LIN {X 85.009,Y 2.500,Z 47.262,A 180.000,B 0.000,C 180.000} C_DIS
LIN {X 84.772,Y 2.500,Z 47.254,A 180.000,B 0.000,C 180.000} C_DIS
LIN {X 84.615,Y 2.500,Z 47.248,A 180.000,B 0.000,C 180.000} C_DIS
LIN {X 84.536,Y 2.500,Z 47.246,A 180.000,B 0.000,C 180.000} C_DIS
LIN {X 84.379,Y 2.500,Z 47.240,A 180.000,B 0.000,C 180.000} C_DIS
LIN {X 84.142,Y 2.500,Z 47.232,A 180.000,B 0.000,C 180.000} C_DIS
LIN {X 83.985,Y 2.500,Z 47.226,A 180.000,B 0.000,C 180.000} C_DIS
LIN {X 83.906,Y 2.500,Z 47.224,A 180.000,B 0.000,C 180.000} C_DIS
LIN {X 83.749,Y 2.500,Z 47.218,A 180.000,B 0.000,C 180.000} C_DIS
LIN {X 83.512,Y 2.500,Z 47.210,A 180.000,B 0.000,C 180.000} C_DIS
LIN {X 83.355,Y 2.500,Z 47.204,A 180.000,B 0.000,C 180.000} C_DIS
LIN {X 83.276,Y 2.500,Z 47.202,A 180.000,B 0.000,C 180.000} C_DIS
LIN {X 83.119,Y 2.500,Z 47.196,A 180.000,B 0.000,C 180.000} C_DIS
LIN {X 82.961,Y 2.500,Z 47.191,A 180.000,B 0.000,C 180.000} C_DIS
LIN {X 82.804,Y 2.500,Z 47.185,A 180.000,B 0.000,C 180.000} C_DIS
LIN {X 82.646,Y 2.500,Z 47.180,A 180.000,B 0.000,C 180.000} C_DIS
LIN {X 82.489,Y 2.500,Z 47.174,A 180.000,B 0.000,C 180.000} C_DIS
LIN {X 82.331,Y 2.500,Z 47.169,A 180.000,B 0.000,C 180.000} C_DIS
LIN {X 82.174,Y 2.500,Z 47.164,A 180.000,B 0.000,C 180.000} C_DIS
LIN {X 82.095,Y 2.500,Z 47.161,A 180.000,B 0.000,C 180.000} C_DIS
LIN {X 82.016,Y 2.500,Z 47.159,A 180.000,B 0.000,C 180.000} C_DIS
LIN {X 81.937,Y 2.500,Z 47.156,A 180.000,B 0.000,C 180.000} C_DIS
LIN {X 81.859,Y 2.500,Z 47.154,A 180.000,B 0.000,C 180.000} C_DIS
LIN {X 81.780,Y 2.500,Z 47.151,A 180.000,B 0.000,C 180.000} C_DIS
LIN {X 81.701,Y 2.500,Z 47.148,A 180.000,B 0.000,C 180.000} C_DIS
LIN {X 81.544,Y 2.500,Z 47.143,A 180.000,B 0.000,C 180.000} C_DIS
LIN {X 81.386,Y 2.500,Z 47.139,A 180.000,B 0.000,C 180.000} C_DIS
LIN {X 81.229,Y 2.500,Z 47.134,A 180.000,B 0.000,C 180.000} C_DIS
LIN {X 81.071,Y 2.500,Z 47.129,A 180.000,B 0.000,C 180.000} C_DIS
LIN {X 80.914,Y 2.500,Z 47.124,A 180.000,B 0.000,C 180.000} C_DIS
LIN {X 80.756,Y 2.500,Z 47.120,A 180.000,B 0.000,C 180.000} C_DIS
LIN {X 80.599,Y 2.500,Z 47.115,A 180.000,B 0.000,C 180.000} C_DIS
LIN {X 80.441,Y 2.500,Z 47.110,A 180.000,B 0.000,C 180.000} C_DIS
LIN {X 80.284,Y 2.500,Z 47.106,A 180.000,B 0.000,C 180.000} C_DIS
LIN {X 80.126,Y 2.500,Z 47.102,A 180.000,B 0.000,C 180.000} C_DIS
LIN {X 79.969,Y 2.500,Z 47.097,A 180.000,B 0.000,C 180.000} C_DIS
LIN {X 79.811,Y 2.500,Z 47.093,A 180.000,B 0.000,C 180.000} C_DIS
LIN {X 79.654,Y 2.500,Z 47.089,A 180.000,B 0.000,C 180.000} C_DIS
LIN {X 79.496,Y 2.500,Z 47.085,A 180.000,B 0.000,C 180.000} C_DIS
LIN {X 79.339,Y 2.500,Z 47.081,A 180.000,B 0.000,C 180.000} C_DIS
LIN {X 79.181,Y 2.500,Z 47.077,A 180.000,B 0.000,C 180.000} C_DIS
LIN {X 79.024,Y 2.500,Z 47.073,A 180.000,B 0.000,C 180.000} C_DIS
LIN {X 78.866,Y 2.500,Z 47.070,A 180.000,B 0.000,C 180.000} C_DIS
LIN {X 78.709,Y 2.500,Z 47.066,A 180.000,B 0.000,C 180.000} C_DIS
LIN {X 78.551,Y 2.500,Z 47.062,A 180.000,B 0.000,C 180.000} C_DIS
LIN {X 78.394,Y 2.500,Z 47.059,A 180.000,B 0.000,C 180.000} C_DIS
LIN {X 78.236,Y 2.500,Z 47.056,A 180.000,B 0.000,C 180.000} C_DIS
LIN {X 78.079,Y 2.500,Z 47.052,A 180.000,B 0.000,C 180.000} C_DIS
LIN {X 77.921,Y 2.500,Z 47.049,A 180.000,B 0.000,C 180.000} C_DIS
LIN {X 77.764,Y 2.500,Z 47.046,A 180.000,B 0.000,C 180.000} C_DIS
LIN {X 77.606,Y 2.500,Z 47.043,A 180.000,B 0.000,C 180.000} C_DIS
LIN {X 77.449,Y 2.500,Z 47.040,A 180.000,B 0.000,C 180.000} C_DIS
LIN {X 77.291,Y 2.500,Z 47.037,A 180.000,B 0.000,C 180.000} C_DIS
LIN {X 77.134,Y 2.500,Z 47.034,A 180.000,B 0.000,C 180.000} C_DIS
LIN {X 76.976,Y 2.500,Z 47.032,A 180.000,B 0.000,C 180.000} C_DIS
LIN {X 76.819,Y 2.500,Z 47.029,A 180.000,B 0.000,C 180.000} C_DIS
LIN {X 76.661,Y 2.500,Z 47.027,A 180.000,B 0.000,C 180.000} C_DIS
LIN {X 76.346,Y 2.500,Z 47.022,A 180.000,B 0.000,C 180.000} C_DIS
LIN {X 76.031,Y 2.500,Z 47.018,A 180.000,B 0.000,C 180.000} C_DIS
LIN {X 75.716,Y 2.500,Z 47.014,A 180.000,B 0.000,C 180.000} C_DIS
LIN {X 75.401,Y 2.500,Z 47.011,A 180.000,B 0.000,C 180.000} C_DIS
LIN {X 75.086,Y 2.500,Z 47.008,A 180.000,B 0.000,C 180.000} C_DIS
LIN {X 74.771,Y 2.500,Z 47.005,A 180.000,B 0.000,C 180.000} C_DIS
LIN {X 74.456,Y 2.500,Z 47.003,A 180.000,B 0.000,C 180.000} C_DIS
LIN {X 74.141,Y 2.500,Z 47.002,A 180.000,B 0.000,C 180.000} C_DIS
LIN {X 73.826,Y 2.500,Z 47.001,A 180.000,B 0.000,C 180.000} C_DIS
LIN {X 73.511,Y 2.500,Z 47.000,A 180.000,B 0.000,C 180.000} C_DIS
LIN {X 73.280,Y 2.500,Z 47.000,A 180.000,B 0.000,C 180.000} C_DIS
; Cutting Move Starts
LIN {X 5.009,Y 2.500,Z 47.000,A 180.000,B 0.000,C 180.000} C_DIS
LIN {X 4.830,Y 2.506,Z 47.000,A 180.000,B 0.000,C 180.000} C_DIS
LIN {X 4.827,Y 2.506,Z 47.000,A 180.000,B 0.000,C 180.000} C_DIS
LIN {X 4.651,Y 2.524,Z 47.000,A 180.000,B 0.000,C 180.000} C_DIS
LIN {X 4.472,Y 2.556,Z 47.000,A 180.000,B 0.000,C 180.000} C_DIS
LIN {X 4.294,Y 2.602,Z 47.000,A 180.000,B 0.000,C 180.000} C_DIS
LIN {X 4.115,Y 2.662,Z 47.000,A 180.000,B 0.000,C 180.000} C_DIS
LIN {X 4.057,Y 2.685,Z 47.000,A 180.000,B 0.000,C 180.000} C_DIS
LIN {X 3.936,Y 2.738,Z 47.000,A 180.000,B 0.000,C 180.000} C_DIS
LIN {X 3.757,Y 2.831,Z 47.000,A 180.000,B 0.000,C 180.000} C_DIS
LIN {X 3.702,Y 2.864,Z 47.000,A 180.000,B 0.000,C 180.000} C_DIS
LIN {X 3.579,Y 2.943,Z 47.000,A 180.000,B 0.000,C 180.000} C_DIS
LIN {X 3.445,Y 3.042,Z 47.000,A 180.000,B 0.000,C 180.000} C_DIS
LIN {X 3.400,Y 3.079,Z 47.000,A 180.000,B 0.000,C 180.000} C_DIS
LIN {X 3.243,Y 3.221,Z 47.000,A 180.000,B 0.000,C 180.000} C_DIS
LIN {X 3.221,Y 3.243,Z 47.000,A 180.000,B 0.000,C 180.000} C_DIS
LIN {X 3.079,Y 3.400,Z 47.000,A 180.000,B 0.000,C 180.000} C_DIS
LIN {X 3.042,Y 3.445,Z 47.000,A 180.000,B 0.000,C 180.000} C_DIS
LIN {X 2.943,Y 3.579,Z 47.000,A 180.000,B 0.000,C 180.000} C_DIS
LIN {X 2.864,Y 3.702,Z 47.000,A 180.000,B 0.000,C 180.000} C_DIS
LIN {X 2.831,Y 3.757,Z 47.000,A 180.000,B 0.000,C 180.000} C_DIS
LIN {X 2.738,Y 3.936,Z 47.000,A 180.000,B 0.000,C 180.000} C_DIS
LIN {X 2.685,Y 4.057,Z 47.000,A 180.000,B 0.000,C 180.000} C_DIS
LIN {X 2.662,Y 4.115,Z 47.000,A 180.000,B 0.000,C 180.000} C_DIS
LIN {X 2.602,Y 4.294,Z 47.000,A 180.000,B 0.000,C 180.000} C_DIS
LIN {X 2.556,Y 4.472,Z 47.000,A 180.000,B 0.000,C 180.000} C_DIS
LIN {X 2.524,Y 4.651,Z 47.000,A 180.000,B 0.000,C 180.000} C_DIS
LIN {X 2.506,Y 4.827,Z 47.000,A 180.000,B 0.000,C 180.000} C_DIS
LIN {X 2.506,Y 4.830,Z 47.000,A 180.000,B 0.000,C 180.000} C_DIS
LIN {X 2.500,Y 5.009,Z 47.000,A 180.000,B 0.000,C 180.000} C_DIS
LIN {X 2.500,Y 149.991,Z 47.000,A 180.000,B 0.000,C 180.000} C_DIS
LIN {X 2.506,Y 150.170,Z 47.000,A 180.000,B 0.000,C 180.000} C_DIS
LIN {X 2.506,Y 150.173,Z 47.000,A 180.000,B 0.000,C 180.000} C_DIS
LIN {X 2.524,Y 150.349,Z 47.000,A 180.000,B 0.000,C 180.000} C_DIS
LIN {X 2.556,Y 150.528,Z 47.000,A 180.000,B 0.000,C 180.000} C_DIS
LIN {X 2.602,Y 150.706,Z 47.000,A 180.000,B 0.000,C 180.000} C_DIS
LIN {X 2.662,Y 150.885,Z 47.000,A 180.000,B 0.000,C 180.000} C_DIS
LIN {X 2.685,Y 150.943,Z 47.000,A 180.000,B 0.000,C 180.000} C_DIS
LIN {X 2.738,Y 151.064,Z 47.000,A 180.000,B 0.000,C 180.000} C_DIS
LIN {X 2.831,Y 151.243,Z 47.000,A 180.000,B 0.000,C 180.000} C_DIS
LIN {X 2.864,Y 151.298,Z 47.000,A 180.000,B 0.000,C 180.000} C_DIS
LIN {X 2.943,Y 151.421,Z 47.000,A 180.000,B 0.000,C 180.000} C_DIS
LIN {X 3.042,Y 151.555,Z 47.000,A 180.000,B 0.000,C 180.000} C_DIS
LIN {X 3.079,Y 151.600,Z 47.000,A 180.000,B 0.000,C 180.000} C_DIS
LIN {X 3.221,Y 151.757,Z 47.000,A 180.000,B 0.000,C 180.000} C_DIS
LIN {X 3.243,Y 151.779,Z 47.000,A 180.000,B 0.000,C 180.000} C_DIS
LIN {X 3.400,Y 151.921,Z 47.000,A 180.000,B 0.000,C 180.000} C_DIS
LIN {X 3.445,Y 151.958,Z 47.000,A 180.000,B 0.000,C 180.000} C_DIS
LIN {X 3.579,Y 152.057,Z 47.000,A 180.000,B 0.000,C 180.000} C_DIS
LIN {X 3.702,Y 152.136,Z 47.000,A 180.000,B 0.000,C 180.000} C_DIS
LIN {X 3.757,Y 152.169,Z 47.000,A 180.000,B 0.000,C 180.000} C_DIS
LIN {X 3.936,Y 152.262,Z 47.000,A 180.000,B 0.000,C 180.000} C_DIS
LIN {X 4.057,Y 152.315,Z 47.000,A 180.000,B 0.000,C 180.000} C_DIS
LIN {X 4.115,Y 152.338,Z 47.000,A 180.000,B 0.000,C 180.000} C_DIS
LIN {X 4.294,Y 152.398,Z 47.000,A 180.000,B 0.000,C 180.000} C_DIS
LIN {X 4.472,Y 152.444,Z 47.000,A 180.000,B 0.000,C 180.000} C_DIS
LIN {X 4.651,Y 152.476,Z 47.000,A 180.000,B 0.000,C 180.000} C_DIS
LIN {X 4.827,Y 152.494,Z 47.000,A 180.000,B 0.000,C 180.000} C_DIS
LIN {X 4.830,Y 152.494,Z 47.000,A 180.000,B 0.000,C 180.000} C_DIS
LIN {X 5.009,Y 152.500,Z 47.000,A 180.000,B 0.000,C 180.000} C_DIS
LIN {X 149.991,Y 152.500,Z 47.000,A 180.000,B 0.000,C 180.000} C_DIS
LIN {X 150.170,Y 152.494,Z 47.000,A 180.000,B 0.000,C 180.000} C_DIS
LIN {X 150.173,Y 152.494,Z 47.000,A 180.000,B 0.000,C 180.000} C_DIS
LIN {X 150.349,Y 152.476,Z 47.000,A 180.000,B 0.000,C 180.000} C_DIS
LIN {X 150.528,Y 152.444,Z 47.000,A 180.000,B 0.000,C 180.000} C_DIS
LIN {X 150.706,Y 152.398,Z 47.000,A 180.000,B 0.000,C 180.000} C_DIS
LIN {X 150.885,Y 152.338,Z 47.000,A 180.000,B 0.000,C 180.000} C_DIS
LIN {X 150.943,Y 152.315,Z 47.000,A 180.000,B 0.000,C 180.000} C_DIS
LIN {X 151.064,Y 152.262,Z 47.000,A 180.000,B 0.000,C 180.000} C_DIS
LIN {X 151.243,Y 152.169,Z 47.000,A 180.000,B 0.000,C 180.000} C_DIS
LIN {X 151.298,Y 152.136,Z 47.000,A 180.000,B 0.000,C 180.000} C_DIS
LIN {X 151.421,Y 152.057,Z 47.000,A 180.000,B 0.000,C 180.000} C_DIS
LIN {X 151.555,Y 151.958,Z 47.000,A 180.000,B 0.000,C 180.000} C_DIS
LIN {X 151.600,Y 151.921,Z 47.000,A 180.000,B 0.000,C 180.000} C_DIS
LIN {X 151.757,Y 151.779,Z 47.000,A 180.000,B 0.000,C 180.000} C_DIS
LIN {X 151.779,Y 151.757,Z 47.000,A 180.000,B 0.000,C 180.000} C_DIS
LIN {X 151.921,Y 151.600,Z 47.000,A 180.000,B 0.000,C 180.000} C_DIS
LIN {X 151.958,Y 151.555,Z 47.000,A 180.000,B 0.000,C 180.000} C_DIS
LIN {X 152.057,Y 151.421,Z 47.000,A 180.000,B 0.000,C 180.000} C_DIS
LIN {X 152.136,Y 151.298,Z 47.000,A 180.000,B 0.000,C 180.000} C_DIS
LIN {X 152.169,Y 151.243,Z 47.000,A 180.000,B 0.000,C 180.000} C_DIS
LIN {X 152.262,Y 151.064,Z 47.000,A 180.000,B 0.000,C 180.000} C_DIS
LIN {X 152.315,Y 150.943,Z 47.000,A 180.000,B 0.000,C 180.000} C_DIS
LIN {X 152.338,Y 150.885,Z 47.000,A 180.000,B 0.000,C 180.000} C_DIS
LIN {X 152.398,Y 150.706,Z 47.000,A 180.000,B 0.000,C 180.000} C_DIS
LIN {X 152.444,Y 150.528,Z 47.000,A 180.000,B 0.000,C 180.000} C_DIS
LIN {X 152.476,Y 150.349,Z 47.000,A 180.000,B 0.000,C 180.000} C_DIS
LIN {X 152.494,Y 150.173,Z 47.000,A 180.000,B 0.000,C 180.000} C_DIS
LIN {X 152.494,Y 150.170,Z 47.000,A 180.000,B 0.000,C 180.000} C_DIS
LIN {X 152.500,Y 149.991,Z 47.000,A 180.000,B 0.000,C 180.000} C_DIS
LIN {X 152.500,Y 5.009,Z 47.000,A 180.000,B 0.000,C 180.000} C_DIS
LIN {X 152.494,Y 4.830,Z 47.000,A 180.000,B 0.000,C 180.000} C_DIS
LIN {X 152.494,Y 4.827,Z 47.000,A 180.000,B 0.000,C 180.000} C_DIS
LIN {X 152.476,Y 4.651,Z 47.000,A 180.000,B 0.000,C 180.000} C_DIS
LIN {X 152.444,Y 4.472,Z 47.000,A 180.000,B 0.000,C 180.000} C_DIS
LIN {X 152.398,Y 4.294,Z 47.000,A 180.000,B 0.000,C 180.000} C_DIS
LIN {X 152.338,Y 4.115,Z 47.000,A 180.000,B 0.000,C 180.000} C_DIS
LIN {X 152.315,Y 4.057,Z 47.000,A 180.000,B 0.000,C 180.000} C_DIS
LIN {X 152.262,Y 3.936,Z 47.000,A 180.000,B 0.000,C 180.000} C_DIS
LIN {X 152.169,Y 3.757,Z 47.000,A 180.000,B 0.000,C 180.000} C_DIS
LIN {X 152.136,Y 3.702,Z 47.000,A 180.000,B 0.000,C 180.000} C_DIS
LIN {X 152.057,Y 3.579,Z 47.000,A 180.000,B 0.000,C 180.000} C_DIS
LIN {X 151.958,Y 3.445,Z 47.000,A 180.000,B 0.000,C 180.000} C_DIS
LIN {X 151.921,Y 3.400,Z 47.000,A 180.000,B 0.000,C 180.000} C_DIS
LIN {X 151.779,Y 3.243,Z 47.000,A 180.000,B 0.000,C 180.000} C_DIS
LIN {X 151.757,Y 3.221,Z 47.000,A 180.000,B 0.000,C 180.000} C_DIS
LIN {X 151.600,Y 3.079,Z 47.000,A 180.000,B 0.000,C 180.000} C_DIS
LIN {X 151.555,Y 3.042,Z 47.000,A 180.000,B 0.000,C 180.000} C_DIS
LIN {X 151.421,Y 2.943,Z 47.000,A 180.000,B 0.000,C 180.000} C_DIS
LIN {X 151.298,Y 2.864,Z 47.000,A 180.000,B 0.000,C 180.000} C_DIS
LIN {X 151.243,Y 2.831,Z 47.000,A 180.000,B 0.000,C 180.000} C_DIS
LIN {X 151.064,Y 2.738,Z 47.000,A 180.000,B 0.000,C 180.000} C_DIS
LIN {X 150.943,Y 2.685,Z 47.000,A 180.000,B 0.000,C 180.000} C_DIS
LIN {X 150.885,Y 2.662,Z 47.000,A 180.000,B 0.000,C 180.000} C_DIS
LIN {X 150.706,Y 2.602,Z 47.000,A 180.000,B 0.000,C 180.000} C_DIS
LIN {X 150.528,Y 2.556,Z 47.000,A 180.000,B 0.000,C 180.000} C_DIS
LIN {X 150.349,Y 2.524,Z 47.000,A 180.000,B 0.000,C 180.000} C_DIS
LIN {X 150.173,Y 2.506,Z 47.000,A 180.000,B 0.000,C 180.000} C_DIS
LIN {X 150.170,Y 2.506,Z 47.000,A 180.000,B 0.000,C 180.000} C_DIS
LIN {X 149.991,Y 2.500,Z 47.000,A 180.000,B 0.000,C 180.000} C_DIS
LIN {X 110.366,Y 2.500,Z 47.000,A 180.000,B 0.000,C 180.000} C_DIS
LIN {X 73.280,Y 2.500,Z 47.000,A 180.000,B 0.000,C 180.000} C_DIS
; Link Move Starts
LIN {X 72.965,Y 2.500,Z 47.000,A 180.000,B 0.000,C 180.000} C_DIS
LIN {X 72.650,Y 2.500,Z 46.999,A 180.000,B 0.000,C 180.000} C_DIS
LIN {X 72.335,Y 2.500,Z 46.998,A 180.000,B 0.000,C 180.000} C_DIS
LIN {X 72.020,Y 2.500,Z 46.996,A 180.000,B 0.000,C 180.000} C_DIS
LIN {X 71.705,Y 2.500,Z 46.994,A 180.000,B 0.000,C 180.000} C_DIS
LIN {X 71.390,Y 2.500,Z 46.991,A 180.000,B 0.000,C 180.000} C_DIS
LIN {X 71.075,Y 2.500,Z 46.988,A 180.000,B 0.000,C 180.000} C_DIS
LIN {X 70.760,Y 2.500,Z 46.985,A 180.000,B 0.000,C 180.000} C_DIS
LIN {X 70.445,Y 2.500,Z 46.981,A 180.000,B 0.000,C 180.000} C_DIS
LIN {X 70.130,Y 2.500,Z 46.977,A 180.000,B 0.000,C 180.000} C_DIS
LIN {X 69.815,Y 2.500,Z 46.972,A 180.000,B 0.000,C 180.000} C_DIS
LIN {X 69.658,Y 2.500,Z 46.969,A 180.000,B 0.000,C 180.000} C_DIS
LIN {X 69.500,Y 2.500,Z 46.967,A 180.000,B 0.000,C 180.000} C_DIS
LIN {X 69.343,Y 2.500,Z 46.964,A 180.000,B 0.000,C 180.000} C_DIS
LIN {X 69.185,Y 2.500,Z 46.961,A 180.000,B 0.000,C 180.000} C_DIS
LIN {X 69.028,Y 2.500,Z 46.959,A 180.000,B 0.000,C 180.000} C_DIS
LIN {X 68.870,Y 2.500,Z 46.956,A 180.000,B 0.000,C 180.000} C_DIS
LIN {X 68.713,Y 2.500,Z 46.952,A 180.000,B 0.000,C 180.000} C_DIS
LIN {X 68.555,Y 2.500,Z 46.949,A 180.000,B 0.000,C 180.000} C_DIS
LIN {X 68.398,Y 2.500,Z 46.946,A 180.000,B 0.000,C 180.000} C_DIS
LIN {X 68.240,Y 2.500,Z 46.943,A 180.000,B 0.000,C 180.000} C_DIS
LIN {X 68.083,Y 2.500,Z 46.939,A 180.000,B 0.000,C 180.000} C_DIS
LIN {X 67.925,Y 2.500,Z 46.936,A 180.000,B 0.000,C 180.000} C_DIS
LIN {X 67.768,Y 2.500,Z 46.932,A 180.000,B 0.000,C 180.000} C_DIS
LIN {X 67.610,Y 2.500,Z 46.928,A 180.000,B 0.000,C 180.000} C_DIS
LIN {X 67.453,Y 2.500,Z 46.925,A 180.000,B 0.000,C 180.000} C_DIS
LIN {X 67.295,Y 2.500,Z 46.921,A 180.000,B 0.000,C 180.000} C_DIS
LIN {X 67.138,Y 2.500,Z 46.917,A 180.000,B 0.000,C 180.000} C_DIS
LIN {X 66.980,Y 2.500,Z 46.913,A 180.000,B 0.000,C 180.000} C_DIS
LIN {X 66.823,Y 2.500,Z 46.909,A 180.000,B 0.000,C 180.000} C_DIS
LIN {X 66.665,Y 2.500,Z 46.905,A 180.000,B 0.000,C 180.000} C_DIS
LIN {X 66.508,Y 2.500,Z 46.900,A 180.000,B 0.000,C 180.000} C_DIS
LIN {X 66.350,Y 2.500,Z 46.896,A 180.000,B 0.000,C 180.000} C_DIS
LIN {X 66.193,Y 2.500,Z 46.892,A 180.000,B 0.000,C 180.000} C_DIS
LIN {X 66.035,Y 2.500,Z 46.887,A 180.000,B 0.000,C 180.000} C_DIS
LIN {X 65.878,Y 2.500,Z 46.883,A 180.000,B 0.000,C 180.000} C_DIS
LIN {X 65.720,Y 2.500,Z 46.878,A 180.000,B 0.000,C 180.000} C_DIS
LIN {X 65.563,Y 2.500,Z 46.873,A 180.000,B 0.000,C 180.000} C_DIS
LIN {X 65.405,Y 2.500,Z 46.869,A 180.000,B 0.000,C 180.000} C_DIS
LIN {X 65.248,Y 2.500,Z 46.864,A 180.000,B 0.000,C 180.000} C_DIS
LIN {X 65.090,Y 2.500,Z 46.859,A 180.000,B 0.000,C 180.000} C_DIS
LIN {X 64.933,Y 2.500,Z 46.854,A 180.000,B 0.000,C 180.000} C_DIS
LIN {X 64.854,Y 2.500,Z 46.851,A 180.000,B 0.000,C 180.000} C_DIS
LIN {X 64.775,Y 2.500,Z 46.849,A 180.000,B 0.000,C 180.000} C_DIS
LIN {X 64.697,Y 2.500,Z 46.846,A 180.000,B 0.000,C 180.000} C_DIS
LIN {X 64.618,Y 2.500,Z 46.844,A 180.000,B 0.000,C 180.000} C_DIS
LIN {X 64.539,Y 2.500,Z 46.841,A 180.000,B 0.000,C 180.000} C_DIS
LIN {X 64.460,Y 2.500,Z 46.839,A 180.000,B 0.000,C 180.000} C_DIS
LIN {X 64.382,Y 2.500,Z 46.836,A 180.000,B 0.000,C 180.000} C_DIS
LIN {X 64.224,Y 2.500,Z 46.831,A 180.000,B 0.000,C 180.000} C_DIS
LIN {X 64.067,Y 2.500,Z 46.825,A 180.000,B 0.000,C 180.000} C_DIS
LIN {X 63.909,Y 2.500,Z 46.820,A 180.000,B 0.000,C 180.000} C_DIS
LIN {X 63.752,Y 2.500,Z 46.815,A 180.000,B 0.000,C 180.000} C_DIS
LIN {X 63.594,Y 2.500,Z 46.809,A 180.000,B 0.000,C 180.000} C_DIS
LIN {X 63.515,Y 2.500,Z 46.806,A 180.000,B 0.000,C 180.000} C_DIS
LIN {X 63.358,Y 2.500,Z 46.801,A 180.000,B 0.000,C 180.000} C_DIS
LIN {X 63.122,Y 2.500,Z 46.793,A 180.000,B 0.000,C 180.000} C_DIS
LIN {X 62.964,Y 2.500,Z 46.787,A 180.000,B 0.000,C 180.000} C_DIS
LIN {X 62.885,Y 2.500,Z 46.785,A 180.000,B 0.000,C 180.000} C_DIS
LIN {X 62.728,Y 2.500,Z 46.779,A 180.000,B 0.000,C 180.000} C_DIS
LIN {X 62.492,Y 2.500,Z 46.771,A 180.000,B 0.000,C 180.000} C_DIS
LIN {X 62.334,Y 2.500,Z 46.765,A 180.000,B 0.000,C 180.000} C_DIS
LIN {X 62.255,Y 2.500,Z 46.763,A 180.000,B 0.000,C 180.000} C_DIS
LIN {X 62.098,Y 2.500,Z 46.757,A 180.000,B 0.000,C 180.000} C_DIS
LIN {X 61.862,Y 2.500,Z 46.749,A 180.000,B 0.000,C 180.000} C_DIS
LIN {X 61.704,Y 2.500,Z 46.743,A 180.000,B 0.000,C 180.000} C_DIS
LIN {X 61.625,Y 2.500,Z 46.741,A 180.000,B 0.000,C 180.000} C_DIS
LIN {X 61.468,Y 2.500,Z 46.735,A 180.000,B 0.000,C 180.000} C_DIS
LIN {X 61.232,Y 2.500,Z 46.727,A 180.000,B 0.000,C 180.000} C_DIS
LIN {X 61.074,Y 2.500,Z 46.721,A 180.000,B 0.000,C 180.000} C_DIS
LIN {X 60.995,Y 2.500,Z 46.719,A 180.000,B 0.000,C 180.000} C_DIS
LIN {X 60.838,Y 2.500,Z 46.713,A 180.000,B 0.000,C 180.000} C_DIS
LIN {X 60.365,Y 2.500,Z 46.697,A 180.000,B 0.000,C 180.000} C_DIS
LIN {X 60.208,Y 2.500,Z 46.691,A 180.000,B 0.000,C 180.000} C_DIS
LIN {X 59.735,Y 2.500,Z 46.675,A 180.000,B 0.000,C 180.000} C_DIS
LIN {X 59.578,Y 2.500,Z 46.669,A 180.000,B 0.000,C 180.000} C_DIS
LIN {X 59.027,Y 2.500,Z 46.650,A 180.000,B 0.000,C 180.000} C_DIS
LIN {X 58.554,Y 2.500,Z 46.633,A 180.000,B 0.000,C 180.000} C_DIS
LIN {X 58.397,Y 2.500,Z 46.628,A 180.000,B 0.000,C 180.000} C_DIS
LIN {X 57.924,Y 2.500,Z 46.611,A 180.000,B 0.000,C 180.000} C_DIS
LIN {X 57.767,Y 2.500,Z 46.606,A 180.000,B 0.000,C 180.000} C_DIS
LIN {X 56.979,Y 2.500,Z 46.578,A 180.000,B 0.000,C 180.000} C_DIS
LIN {X 56.585,Y 2.500,Z 46.565,A 180.000,B 0.000,C 180.000} C_DIS
LIN {X 56.113,Y 2.500,Z 46.548,A 180.000,B 0.000,C 180.000} C_DIS
LIN {X 54.302,Y 2.500,Z 46.485,A 180.000,B 0.000,C 180.000} C_DIS
LIN {X 51.309,Y 2.500,Z 46.380,A 180.000,B 0.000,C 180.000} C_DIS
LIN {X 51.152,Y 2.500,Z 46.375,A 180.000,B 0.000,C 180.000} C_DIS
LIN {X 50.679,Y 2.500,Z 46.358,A 180.000,B 0.000,C 180.000} C_DIS
LIN {X 50.522,Y 2.500,Z 46.353,A 180.000,B 0.000,C 180.000} C_DIS
LIN {X 50.049,Y 2.500,Z 46.336,A 180.000,B 0.000,C 180.000} C_DIS
LIN {X 49.970,Y 2.500,Z 46.334,A 180.000,B 0.000,C 180.000} C_DIS
LIN {X 49.813,Y 2.500,Z 46.328,A 180.000,B 0.000,C 180.000} C_DIS
LIN {X 49.340,Y 2.500,Z 46.312,A 180.000,B 0.000,C 180.000} C_DIS
LIN {X 49.183,Y 2.500,Z 46.306,A 180.000,B 0.000,C 180.000} C_DIS
LIN {X 48.710,Y 2.500,Z 46.290,A 180.000,B 0.000,C 180.000} C_DIS
LIN {X 48.553,Y 2.500,Z 46.284,A 180.000,B 0.000,C 180.000} C_DIS
LIN {X 48.317,Y 2.500,Z 46.276,A 180.000,B 0.000,C 180.000} C_DIS
LIN {X 48.159,Y 2.500,Z 46.270,A 180.000,B 0.000,C 180.000} C_DIS
LIN {X 48.080,Y 2.500,Z 46.268,A 180.000,B 0.000,C 180.000} C_DIS
LIN {X 47.923,Y 2.500,Z 46.262,A 180.000,B 0.000,C 180.000} C_DIS
LIN {X 47.687,Y 2.500,Z 46.254,A 180.000,B 0.000,C 180.000} C_DIS
LIN {X 47.529,Y 2.500,Z 46.248,A 180.000,B 0.000,C 180.000} C_DIS
LIN {X 47.450,Y 2.500,Z 46.246,A 180.000,B 0.000,C 180.000} C_DIS
LIN {X 47.293,Y 2.500,Z 46.240,A 180.000,B 0.000,C 180.000} C_DIS
LIN {X 47.057,Y 2.500,Z 46.232,A 180.000,B 0.000,C 180.000} C_DIS
LIN {X 46.899,Y 2.500,Z 46.226,A 180.000,B 0.000,C 180.000} C_DIS
LIN {X 46.820,Y 2.500,Z 46.224,A 180.000,B 0.000,C 180.000} C_DIS
LIN {X 46.663,Y 2.500,Z 46.218,A 180.000,B 0.000,C 180.000} C_DIS
LIN {X 46.427,Y 2.500,Z 46.210,A 180.000,B 0.000,C 180.000} C_DIS
LIN {X 46.269,Y 2.500,Z 46.204,A 180.000,B 0.000,C 180.000} C_DIS
LIN {X 46.190,Y 2.500,Z 46.202,A 180.000,B 0.000,C 180.000} C_DIS
LIN {X 46.033,Y 2.500,Z 46.196,A 180.000,B 0.000,C 180.000} C_DIS
LIN {X 45.875,Y 2.500,Z 46.191,A 180.000,B 0.000,C 180.000} C_DIS
LIN {X 45.718,Y 2.500,Z 46.185,A 180.000,B 0.000,C 180.000} C_DIS
LIN {X 45.561,Y 2.500,Z 46.180,A 180.000,B 0.000,C 180.000} C_DIS
LIN {X 45.403,Y 2.500,Z 46.174,A 180.000,B 0.000,C 180.000} C_DIS
LIN {X 45.246,Y 2.500,Z 46.169,A 180.000,B 0.000,C 180.000} C_DIS
LIN {X 45.088,Y 2.500,Z 46.164,A 180.000,B 0.000,C 180.000} C_DIS
LIN {X 45.009,Y 2.500,Z 46.161,A 180.000,B 0.000,C 180.000} C_DIS
LIN {X 44.931,Y 2.500,Z 46.159,A 180.000,B 0.000,C 180.000} C_DIS
LIN {X 44.852,Y 2.500,Z 46.156,A 180.000,B 0.000,C 180.000} C_DIS
LIN {X 44.773,Y 2.500,Z 46.154,A 180.000,B 0.000,C 180.000} C_DIS
LIN {X 44.694,Y 2.500,Z 46.151,A 180.000,B 0.000,C 180.000} C_DIS
LIN {X 44.616,Y 2.500,Z 46.148,A 180.000,B 0.000,C 180.000} C_DIS
LIN {X 44.458,Y 2.500,Z 46.143,A 180.000,B 0.000,C 180.000} C_DIS
LIN {X 44.301,Y 2.500,Z 46.139,A 180.000,B 0.000,C 180.000} C_DIS
LIN {X 44.143,Y 2.500,Z 46.134,A 180.000,B 0.000,C 180.000} C_DIS
LIN {X 43.986,Y 2.500,Z 46.129,A 180.000,B 0.000,C 180.000} C_DIS
LIN {X 43.828,Y 2.500,Z 46.124,A 180.000,B 0.000,C 180.000} C_DIS
LIN {X 43.671,Y 2.500,Z 46.120,A 180.000,B 0.000,C 180.000} C_DIS
LIN {X 43.513,Y 2.500,Z 46.115,A 180.000,B 0.000,C 180.000} C_DIS
LIN {X 43.356,Y 2.500,Z 46.110,A 180.000,B 0.000,C 180.000} C_DIS
LIN {X 43.198,Y 2.500,Z 46.106,A 180.000,B 0.000,C 180.000} C_DIS
LIN {X 43.041,Y 2.500,Z 46.102,A 180.000,B 0.000,C 180.000} C_DIS
LIN {X 42.883,Y 2.500,Z 46.097,A 180.000,B 0.000,C 180.000} C_DIS
LIN {X 42.726,Y 2.500,Z 46.093,A 180.000,B 0.000,C 180.000} C_DIS
LIN {X 42.568,Y 2.500,Z 46.089,A 180.000,B 0.000,C 180.000} C_DIS
LIN {X 42.411,Y 2.500,Z 46.085,A 180.000,B 0.000,C 180.000} C_DIS
LIN {X 42.253,Y 2.500,Z 46.081,A 180.000,B 0.000,C 180.000} C_DIS
LIN {X 42.096,Y 2.500,Z 46.077,A 180.000,B 0.000,C 180.000} C_DIS
LIN {X 41.938,Y 2.500,Z 46.073,A 180.000,B 0.000,C 180.000} C_DIS
LIN {X 41.781,Y 2.500,Z 46.070,A 180.000,B 0.000,C 180.000} C_DIS
LIN {X 41.623,Y 2.500,Z 46.066,A 180.000,B 0.000,C 180.000} C_DIS
LIN {X 41.466,Y 2.500,Z 46.062,A 180.000,B 0.000,C 180.000} C_DIS
LIN {X 41.308,Y 2.500,Z 46.059,A 180.000,B 0.000,C 180.000} C_DIS
LIN {X 41.151,Y 2.500,Z 46.056,A 180.000,B 0.000,C 180.000} C_DIS
LIN {X 40.993,Y 2.500,Z 46.052,A 180.000,B 0.000,C 180.000} C_DIS
LIN {X 40.836,Y 2.500,Z 46.049,A 180.000,B 0.000,C 180.000} C_DIS
LIN {X 40.678,Y 2.500,Z 46.046,A 180.000,B 0.000,C 180.000} C_DIS
LIN {X 40.521,Y 2.500,Z 46.043,A 180.000,B 0.000,C 180.000} C_DIS
LIN {X 40.363,Y 2.500,Z 46.040,A 180.000,B 0.000,C 180.000} C_DIS
LIN {X 40.206,Y 2.500,Z 46.037,A 180.000,B 0.000,C 180.000} C_DIS
LIN {X 40.048,Y 2.500,Z 46.034,A 180.000,B 0.000,C 180.000} C_DIS
LIN {X 39.891,Y 2.500,Z 46.032,A 180.000,B 0.000,C 180.000} C_DIS
LIN {X 39.733,Y 2.500,Z 46.029,A 180.000,B 0.000,C 180.000} C_DIS
LIN {X 39.576,Y 2.500,Z 46.027,A 180.000,B 0.000,C 180.000} C_DIS
LIN {X 39.261,Y 2.500,Z 46.022,A 180.000,B 0.000,C 180.000} C_DIS
LIN {X 38.946,Y 2.500,Z 46.018,A 180.000,B 0.000,C 180.000} C_DIS
LIN {X 38.631,Y 2.500,Z 46.014,A 180.000,B 0.000,C 180.000} C_DIS
LIN {X 38.316,Y 2.500,Z 46.011,A 180.000,B 0.000,C 180.000} C_DIS
LIN {X 38.001,Y 2.500,Z 46.008,A 180.000,B 0.000,C 180.000} C_DIS
LIN {X 37.686,Y 2.500,Z 46.005,A 180.000,B 0.000,C 180.000} C_DIS
LIN {X 37.371,Y 2.500,Z 46.003,A 180.000,B 0.000,C 180.000} C_DIS
LIN {X 37.056,Y 2.500,Z 46.002,A 180.000,B 0.000,C 180.000} C_DIS
LIN {X 36.741,Y 2.500,Z 46.001,A 180.000,B 0.000,C 180.000} C_DIS
LIN {X 36.426,Y 2.500,Z 46.000,A 180.000,B 0.000,C 180.000} C_DIS
LIN {X 36.195,Y 2.500,Z 46.000,A 180.000,B 0.000,C 180.000} C_DIS
; Cutting Move Starts
LIN {X 5.009,Y 2.500,Z 46.000,A 180.000,B 0.000,C 180.000} C_DIS
LIN {X 4.830,Y 2.506,Z 46.000,A 180.000,B 0.000,C 180.000} C_DIS
LIN {X 4.827,Y 2.506,Z 46.000,A 180.000,B 0.000,C 180.000} C_DIS
LIN {X 4.651,Y 2.524,Z 46.000,A 180.000,B 0.000,C 180.000} C_DIS
LIN {X 4.472,Y 2.556,Z 46.000,A 180.000,B 0.000,C 180.000} C_DIS
LIN {X 4.294,Y 2.602,Z 46.000,A 180.000,B 0.000,C 180.000} C_DIS
LIN {X 4.115,Y 2.662,Z 46.000,A 180.000,B 0.000,C 180.000} C_DIS
LIN {X 4.057,Y 2.685,Z 46.000,A 180.000,B 0.000,C 180.000} C_DIS
LIN {X 3.936,Y 2.738,Z 46.000,A 180.000,B 0.000,C 180.000} C_DIS
LIN {X 3.757,Y 2.831,Z 46.000,A 180.000,B 0.000,C 180.000} C_DIS
LIN {X 3.702,Y 2.864,Z 46.000,A 180.000,B 0.000,C 180.000} C_DIS
LIN {X 3.579,Y 2.943,Z 46.000,A 180.000,B 0.000,C 180.000} C_DIS
LIN {X 3.445,Y 3.042,Z 46.000,A 180.000,B 0.000,C 180.000} C_DIS
LIN {X 3.400,Y 3.079,Z 46.000,A 180.000,B 0.000,C 180.000} C_DIS
LIN {X 3.243,Y 3.221,Z 46.000,A 180.000,B 0.000,C 180.000} C_DIS
LIN {X 3.221,Y 3.243,Z 46.000,A 180.000,B 0.000,C 180.000} C_DIS
LIN {X 3.079,Y 3.400,Z 46.000,A 180.000,B 0.000,C 180.000} C_DIS
LIN {X 3.042,Y 3.445,Z 46.000,A 180.000,B 0.000,C 180.000} C_DIS
LIN {X 2.943,Y 3.579,Z 46.000,A 180.000,B 0.000,C 180.000} C_DIS
LIN {X 2.864,Y 3.702,Z 46.000,A 180.000,B 0.000,C 180.000} C_DIS
LIN {X 2.831,Y 3.757,Z 46.000,A 180.000,B 0.000,C 180.000} C_DIS
LIN {X 2.738,Y 3.936,Z 46.000,A 180.000,B 0.000,C 180.000} C_DIS
LIN {X 2.685,Y 4.057,Z 46.000,A 180.000,B 0.000,C 180.000} C_DIS
LIN {X 2.662,Y 4.115,Z 46.000,A 180.000,B 0.000,C 180.000} C_DIS
LIN {X 2.602,Y 4.294,Z 46.000,A 180.000,B 0.000,C 180.000} C_DIS
LIN {X 2.556,Y 4.472,Z 46.000,A 180.000,B 0.000,C 180.000} C_DIS
LIN {X 2.524,Y 4.651,Z 46.000,A 180.000,B 0.000,C 180.000} C_DIS
LIN {X 2.506,Y 4.827,Z 46.000,A 180.000,B 0.000,C 180.000} C_DIS
LIN {X 2.506,Y 4.830,Z 46.000,A 180.000,B 0.000,C 180.000} C_DIS
LIN {X 2.500,Y 5.009,Z 46.000,A 180.000,B 0.000,C 180.000} C_DIS
LIN {X 2.500,Y 149.991,Z 46.000,A 180.000,B 0.000,C 180.000} C_DIS
LIN {X 2.506,Y 150.170,Z 46.000,A 180.000,B 0.000,C 180.000} C_DIS
LIN {X 2.506,Y 150.173,Z 46.000,A 180.000,B 0.000,C 180.000} C_DIS
LIN {X 2.524,Y 150.349,Z 46.000,A 180.000,B 0.000,C 180.000} C_DIS
LIN {X 2.556,Y 150.528,Z 46.000,A 180.000,B 0.000,C 180.000} C_DIS
LIN {X 2.602,Y 150.706,Z 46.000,A 180.000,B 0.000,C 180.000} C_DIS
LIN {X 2.662,Y 150.885,Z 46.000,A 180.000,B 0.000,C 180.000} C_DIS
LIN {X 2.685,Y 150.943,Z 46.000,A 180.000,B 0.000,C 180.000} C_DIS
LIN {X 2.738,Y 151.064,Z 46.000,A 180.000,B 0.000,C 180.000} C_DIS
LIN {X 2.831,Y 151.243,Z 46.000,A 180.000,B 0.000,C 180.000} C_DIS
LIN {X 2.864,Y 151.298,Z 46.000,A 180.000,B 0.000,C 180.000} C_DIS
LIN {X 2.943,Y 151.421,Z 46.000,A 180.000,B 0.000,C 180.000} C_DIS
LIN {X 3.042,Y 151.555,Z 46.000,A 180.000,B 0.000,C 180.000} C_DIS
LIN {X 3.079,Y 151.600,Z 46.000,A 180.000,B 0.000,C 180.000} C_DIS
LIN {X 3.221,Y 151.757,Z 46.000,A 180.000,B 0.000,C 180.000} C_DIS
LIN {X 3.243,Y 151.779,Z 46.000,A 180.000,B 0.000,C 180.000} C_DIS
LIN {X 3.400,Y 151.921,Z 46.000,A 180.000,B 0.000,C 180.000} C_DIS
LIN {X 3.445,Y 151.958,Z 46.000,A 180.000,B 0.000,C 180.000} C_DIS
LIN {X 3.579,Y 152.057,Z 46.000,A 180.000,B 0.000,C 180.000} C_DIS
LIN {X 3.702,Y 152.136,Z 46.000,A 180.000,B 0.000,C 180.000} C_DIS
LIN {X 3.757,Y 152.169,Z 46.000,A 180.000,B 0.000,C 180.000} C_DIS
LIN {X 3.936,Y 152.262,Z 46.000,A 180.000,B 0.000,C 180.000} C_DIS
LIN {X 4.057,Y 152.315,Z 46.000,A 180.000,B 0.000,C 180.000} C_DIS
LIN {X 4.115,Y 152.338,Z 46.000,A 180.000,B 0.000,C 180.000} C_DIS
LIN {X 4.294,Y 152.398,Z 46.000,A 180.000,B 0.000,C 180.000} C_DIS
LIN {X 4.472,Y 152.444,Z 46.000,A 180.000,B 0.000,C 180.000} C_DIS
LIN {X 4.651,Y 152.476,Z 46.000,A 180.000,B 0.000,C 180.000} C_DIS
LIN {X 4.827,Y 152.494,Z 46.000,A 180.000,B 0.000,C 180.000} C_DIS
LIN {X 4.830,Y 152.494,Z 46.000,A 180.000,B 0.000,C 180.000} C_DIS
LIN {X 5.009,Y 152.500,Z 46.000,A 180.000,B 0.000,C 180.000} C_DIS
LIN {X 149.991,Y 152.500,Z 46.000,A 180.000,B 0.000,C 180.000} C_DIS
LIN {X 150.170,Y 152.494,Z 46.000,A 180.000,B 0.000,C 180.000} C_DIS
LIN {X 150.173,Y 152.494,Z 46.000,A 180.000,B 0.000,C 180.000} C_DIS
LIN {X 150.349,Y 152.476,Z 46.000,A 180.000,B 0.000,C 180.000} C_DIS
LIN {X 150.528,Y 152.444,Z 46.000,A 180.000,B 0.000,C 180.000} C_DIS
LIN {X 150.706,Y 152.398,Z 46.000,A 180.000,B 0.000,C 180.000} C_DIS
LIN {X 150.885,Y 152.338,Z 46.000,A 180.000,B 0.000,C 180.000} C_DIS
LIN {X 150.943,Y 152.315,Z 46.000,A 180.000,B 0.000,C 180.000} C_DIS
LIN {X 151.064,Y 152.262,Z 46.000,A 180.000,B 0.000,C 180.000} C_DIS
LIN {X 151.243,Y 152.169,Z 46.000,A 180.000,B 0.000,C 180.000} C_DIS
LIN {X 151.298,Y 152.136,Z 46.000,A 180.000,B 0.000,C 180.000} C_DIS
LIN {X 151.421,Y 152.057,Z 46.000,A 180.000,B 0.000,C 180.000} C_DIS
LIN {X 151.555,Y 151.958,Z 46.000,A 180.000,B 0.000,C 180.000} C_DIS
LIN {X 151.600,Y 151.921,Z 46.000,A 180.000,B 0.000,C 180.000} C_DIS
LIN {X 151.757,Y 151.779,Z 46.000,A 180.000,B 0.000,C 180.000} C_DIS
LIN {X 151.779,Y 151.757,Z 46.000,A 180.000,B 0.000,C 180.000} C_DIS
LIN {X 151.921,Y 151.600,Z 46.000,A 180.000,B 0.000,C 180.000} C_DIS
LIN {X 151.958,Y 151.555,Z 46.000,A 180.000,B 0.000,C 180.000} C_DIS
LIN {X 152.057,Y 151.421,Z 46.000,A 180.000,B 0.000,C 180.000} C_DIS
LIN {X 152.136,Y 151.298,Z 46.000,A 180.000,B 0.000,C 180.000} C_DIS
LIN {X 152.169,Y 151.243,Z 46.000,A 180.000,B 0.000,C 180.000} C_DIS
LIN {X 152.262,Y 151.064,Z 46.000,A 180.000,B 0.000,C 180.000} C_DIS
LIN {X 152.315,Y 150.943,Z 46.000,A 180.000,B 0.000,C 180.000} C_DIS
LIN {X 152.338,Y 150.885,Z 46.000,A 180.000,B 0.000,C 180.000} C_DIS
LIN {X 152.398,Y 150.706,Z 46.000,A 180.000,B 0.000,C 180.000} C_DIS
LIN {X 152.444,Y 150.528,Z 46.000,A 180.000,B 0.000,C 180.000} C_DIS
LIN {X 152.476,Y 150.349,Z 46.000,A 180.000,B 0.000,C 180.000} C_DIS
LIN {X 152.494,Y 150.173,Z 46.000,A 180.000,B 0.000,C 180.000} C_DIS
LIN {X 152.494,Y 150.170,Z 46.000,A 180.000,B 0.000,C 180.000} C_DIS
LIN {X 152.500,Y 149.991,Z 46.000,A 180.000,B 0.000,C 180.000} C_DIS
LIN {X 152.500,Y 5.009,Z 46.000,A 180.000,B 0.000,C 180.000} C_DIS
LIN {X 152.494,Y 4.830,Z 46.000,A 180.000,B 0.000,C 180.000} C_DIS
LIN {X 152.494,Y 4.827,Z 46.000,A 180.000,B 0.000,C 180.000} C_DIS
LIN {X 152.476,Y 4.651,Z 46.000,A 180.000,B 0.000,C 180.000} C_DIS
LIN {X 152.444,Y 4.472,Z 46.000,A 180.000,B 0.000,C 180.000} C_DIS
LIN {X 152.398,Y 4.294,Z 46.000,A 180.000,B 0.000,C 180.000} C_DIS
LIN {X 152.338,Y 4.115,Z 46.000,A 180.000,B 0.000,C 180.000} C_DIS
LIN {X 152.315,Y 4.057,Z 46.000,A 180.000,B 0.000,C 180.000} C_DIS
LIN {X 152.262,Y 3.936,Z 46.000,A 180.000,B 0.000,C 180.000} C_DIS
LIN {X 152.169,Y 3.757,Z 46.000,A 180.000,B 0.000,C 180.000} C_DIS
LIN {X 152.136,Y 3.702,Z 46.000,A 180.000,B 0.000,C 180.000} C_DIS
LIN {X 152.057,Y 3.579,Z 46.000,A 180.000,B 0.000,C 180.000} C_DIS
LIN {X 151.958,Y 3.445,Z 46.000,A 180.000,B 0.000,C 180.000} C_DIS
LIN {X 151.921,Y 3.400,Z 46.000,A 180.000,B 0.000,C 180.000} C_DIS
LIN {X 151.779,Y 3.243,Z 46.000,A 180.000,B 0.000,C 180.000} C_DIS
LIN {X 151.757,Y 3.221,Z 46.000,A 180.000,B 0.000,C 180.000} C_DIS
LIN {X 151.600,Y 3.079,Z 46.000,A 180.000,B 0.000,C 180.000} C_DIS
LIN {X 151.555,Y 3.042,Z 46.000,A 180.000,B 0.000,C 180.000} C_DIS
LIN {X 151.421,Y 2.943,Z 46.000,A 180.000,B 0.000,C 180.000} C_DIS
LIN {X 151.298,Y 2.864,Z 46.000,A 180.000,B 0.000,C 180.000} C_DIS
LIN {X 151.243,Y 2.831,Z 46.000,A 180.000,B 0.000,C 180.000} C_DIS
LIN {X 151.064,Y 2.738,Z 46.000,A 180.000,B 0.000,C 180.000} C_DIS
LIN {X 150.943,Y 2.685,Z 46.000,A 180.000,B 0.000,C 180.000} C_DIS
LIN {X 150.885,Y 2.662,Z 46.000,A 180.000,B 0.000,C 180.000} C_DIS
LIN {X 150.706,Y 2.602,Z 46.000,A 180.000,B 0.000,C 180.000} C_DIS
LIN {X 150.528,Y 2.556,Z 46.000,A 180.000,B 0.000,C 180.000} C_DIS
LIN {X 150.349,Y 2.524,Z 46.000,A 180.000,B 0.000,C 180.000} C_DIS
LIN {X 150.173,Y 2.506,Z 46.000,A 180.000,B 0.000,C 180.000} C_DIS
LIN {X 150.170,Y 2.506,Z 46.000,A 180.000,B 0.000,C 180.000} C_DIS
LIN {X 149.991,Y 2.500,Z 46.000,A 180.000,B 0.000,C 180.000} C_DIS
LIN {X 73.280,Y 2.500,Z 46.000,A 180.000,B 0.000,C 180.000} C_DIS
LIN {X 36.195,Y 2.500,Z 46.000,A 180.000,B 0.000,C 180.000} C_DIS
; Link Move Starts
LIN {X 35.880,Y 2.500,Z 46.000,A 180.000,B 0.000,C 180.000} C_DIS
LIN {X 35.565,Y 2.500,Z 45.999,A 180.000,B 0.000,C 180.000} C_DIS
LIN {X 35.250,Y 2.500,Z 45.998,A 180.000,B 0.000,C 180.000} C_DIS
LIN {X 34.935,Y 2.500,Z 45.996,A 180.000,B 0.000,C 180.000} C_DIS
LIN {X 34.620,Y 2.500,Z 45.994,A 180.000,B 0.000,C 180.000} C_DIS
LIN {X 34.305,Y 2.500,Z 45.991,A 180.000,B 0.000,C 180.000} C_DIS
LIN {X 33.990,Y 2.500,Z 45.988,A 180.000,B 0.000,C 180.000} C_DIS
LIN {X 33.675,Y 2.500,Z 45.985,A 180.000,B 0.000,C 180.000} C_DIS
LIN {X 33.360,Y 2.500,Z 45.981,A 180.000,B 0.000,C 180.000} C_DIS
LIN {X 33.045,Y 2.500,Z 45.977,A 180.000,B 0.000,C 180.000} C_DIS
LIN {X 32.730,Y 2.500,Z 45.972,A 180.000,B 0.000,C 180.000} C_DIS
LIN {X 32.572,Y 2.500,Z 45.969,A 180.000,B 0.000,C 180.000} C_DIS
LIN {X 32.415,Y 2.500,Z 45.967,A 180.000,B 0.000,C 180.000} C_DIS
LIN {X 32.257,Y 2.500,Z 45.964,A 180.000,B 0.000,C 180.000} C_DIS
LIN {X 32.100,Y 2.500,Z 45.961,A 180.000,B 0.000,C 180.000} C_DIS
LIN {X 31.942,Y 2.500,Z 45.959,A 180.000,B 0.000,C 180.000} C_DIS
LIN {X 31.785,Y 2.500,Z 45.956,A 180.000,B 0.000,C 180.000} C_DIS
LIN {X 31.627,Y 2.500,Z 45.952,A 180.000,B 0.000,C 180.000} C_DIS
LIN {X 31.470,Y 2.500,Z 45.949,A 180.000,B 0.000,C 180.000} C_DIS
LIN {X 31.312,Y 2.500,Z 45.946,A 180.000,B 0.000,C 180.000} C_DIS
LIN {X 31.155,Y 2.500,Z 45.943,A 180.000,B 0.000,C 180.000} C_DIS
LIN {X 30.997,Y 2.500,Z 45.939,A 180.000,B 0.000,C 180.000} C_DIS
LIN {X 30.840,Y 2.500,Z 45.936,A 180.000,B 0.000,C 180.000} C_DIS
LIN {X 30.682,Y 2.500,Z 45.932,A 180.000,B 0.000,C 180.000} C_DIS
LIN {X 30.525,Y 2.500,Z 45.928,A 180.000,B 0.000,C 180.000} C_DIS
LIN {X 30.367,Y 2.500,Z 45.925,A 180.000,B 0.000,C 180.000} C_DIS
LIN {X 30.210,Y 2.500,Z 45.921,A 180.000,B 0.000,C 180.000} C_DIS
LIN {X 30.052,Y 2.500,Z 45.917,A 180.000,B 0.000,C 180.000} C_DIS
LIN {X 29.895,Y 2.500,Z 45.913,A 180.000,B 0.000,C 180.000} C_DIS
LIN {X 29.737,Y 2.500,Z 45.909,A 180.000,B 0.000,C 180.000} C_DIS
LIN {X 29.580,Y 2.500,Z 45.905,A 180.000,B 0.000,C 180.000} C_DIS
LIN {X 29.422,Y 2.500,Z 45.900,A 180.000,B 0.000,C 180.000} C_DIS
LIN {X 29.265,Y 2.500,Z 45.896,A 180.000,B 0.000,C 180.000} C_DIS
LIN {X 29.107,Y 2.500,Z 45.892,A 180.000,B 0.000,C 180.000} C_DIS
LIN {X 28.950,Y 2.500,Z 45.887,A 180.000,B 0.000,C 180.000} C_DIS
LIN {X 28.792,Y 2.500,Z 45.883,A 180.000,B 0.000,C 180.000} C_DIS
LIN {X 28.635,Y 2.500,Z 45.878,A 180.000,B 0.000,C 180.000} C_DIS
LIN {X 28.477,Y 2.500,Z 45.873,A 180.000,B 0.000,C 180.000} C_DIS
LIN {X 28.320,Y 2.500,Z 45.869,A 180.000,B 0.000,C 180.000} C_DIS
LIN {X 28.162,Y 2.500,Z 45.864,A 180.000,B 0.000,C 180.000} C_DIS
LIN {X 28.005,Y 2.500,Z 45.859,A 180.000,B 0.000,C 180.000} C_DIS
LIN {X 27.847,Y 2.500,Z 45.854,A 180.000,B 0.000,C 180.000} C_DIS
LIN {X 27.768,Y 2.500,Z 45.851,A 180.000,B 0.000,C 180.000} C_DIS
LIN {X 27.690,Y 2.500,Z 45.849,A 180.000,B 0.000,C 180.000} C_DIS
LIN {X 27.611,Y 2.500,Z 45.846,A 180.000,B 0.000,C 180.000} C_DIS
LIN {X 27.532,Y 2.500,Z 45.844,A 180.000,B 0.000,C 180.000} C_DIS
LIN {X 27.453,Y 2.500,Z 45.841,A 180.000,B 0.000,C 180.000} C_DIS
LIN {X 27.375,Y 2.500,Z 45.839,A 180.000,B 0.000,C 180.000} C_DIS
LIN {X 27.296,Y 2.500,Z 45.836,A 180.000,B 0.000,C 180.000} C_DIS
LIN {X 27.138,Y 2.500,Z 45.831,A 180.000,B 0.000,C 180.000} C_DIS
LIN {X 26.981,Y 2.500,Z 45.825,A 180.000,B 0.000,C 180.000} C_DIS
LIN {X 26.823,Y 2.500,Z 45.820,A 180.000,B 0.000,C 180.000} C_DIS
LIN {X 26.666,Y 2.500,Z 45.815,A 180.000,B 0.000,C 180.000} C_DIS
LIN {X 26.508,Y 2.500,Z 45.809,A 180.000,B 0.000,C 180.000} C_DIS
LIN {X 26.430,Y 2.500,Z 45.806,A 180.000,B 0.000,C 180.000} C_DIS
LIN {X 26.272,Y 2.500,Z 45.801,A 180.000,B 0.000,C 180.000} C_DIS
LIN {X 26.036,Y 2.500,Z 45.793,A 180.000,B 0.000,C 180.000} C_DIS
LIN {X 25.878,Y 2.500,Z 45.787,A 180.000,B 0.000,C 180.000} C_DIS
LIN {X 25.800,Y 2.500,Z 45.785,A 180.000,B 0.000,C 180.000} C_DIS
LIN {X 25.642,Y 2.500,Z 45.779,A 180.000,B 0.000,C 180.000} C_DIS
LIN {X 25.406,Y 2.500,Z 45.771,A 180.000,B 0.000,C 180.000} C_DIS
LIN {X 25.248,Y 2.500,Z 45.765,A 180.000,B 0.000,C 180.000} C_DIS
LIN {X 25.170,Y 2.500,Z 45.763,A 180.000,B 0.000,C 180.000} C_DIS
LIN {X 25.012,Y 2.500,Z 45.757,A 180.000,B 0.000,C 180.000} C_DIS
LIN {X 24.776,Y 2.500,Z 45.749,A 180.000,B 0.000,C 180.000} C_DIS
LIN {X 24.618,Y 2.500,Z 45.743,A 180.000,B 0.000,C 180.000} C_DIS
LIN {X 24.540,Y 2.500,Z 45.741,A 180.000,B 0.000,C 180.000} C_DIS
LIN {X 24.382,Y 2.500,Z 45.735,A 180.000,B 0.000,C 180.000} C_DIS
LIN {X 24.146,Y 2.500,Z 45.727,A 180.000,B 0.000,C 180.000} C_DIS
LIN {X 23.988,Y 2.500,Z 45.721,A 180.000,B 0.000,C 180.000} C_DIS
LIN {X 23.910,Y 2.500,Z 45.719,A 180.000,B 0.000,C 180.000} C_DIS
LIN {X 23.752,Y 2.500,Z 45.713,A 180.000,B 0.000,C 180.000} C_DIS
LIN {X 23.280,Y 2.500,Z 45.697,A 180.000,B 0.000,C 180.000} C_DIS
LIN {X 23.122,Y 2.500,Z 45.691,A 180.000,B 0.000,C 180.000} C_DIS
LIN {X 22.650,Y 2.500,Z 45.675,A 180.000,B 0.000,C 180.000} C_DIS
LIN {X 22.492,Y 2.500,Z 45.669,A 180.000,B 0.000,C 180.000} C_DIS
LIN {X 21.941,Y 2.500,Z 45.650,A 180.000,B 0.000,C 180.000} C_DIS
LIN {X 21.468,Y 2.500,Z 45.633,A 180.000,B 0.000,C 180.000} C_DIS
LIN {X 21.311,Y 2.500,Z 45.628,A 180.000,B 0.000,C 180.000} C_DIS
LIN {X 20.838,Y 2.500,Z 45.611,A 180.000,B 0.000,C 180.000} C_DIS
LIN {X 20.681,Y 2.500,Z 45.606,A 180.000,B 0.000,C 180.000} C_DIS
LIN {X 19.893,Y 2.500,Z 45.578,A 180.000,B 0.000,C 180.000} C_DIS
LIN {X 19.500,Y 2.500,Z 45.565,A 180.000,B 0.000,C 180.000} C_DIS
LIN {X 19.027,Y 2.500,Z 45.548,A 180.000,B 0.000,C 180.000} C_DIS
LIN {X 17.216,Y 2.500,Z 45.485,A 180.000,B 0.000,C 180.000} C_DIS
LIN {X 14.223,Y 2.500,Z 45.380,A 180.000,B 0.000,C 180.000} C_DIS
LIN {X 14.066,Y 2.500,Z 45.375,A 180.000,B 0.000,C 180.000} C_DIS
LIN {X 13.593,Y 2.500,Z 45.358,A 180.000,B 0.000,C 180.000} C_DIS
LIN {X 13.436,Y 2.500,Z 45.353,A 180.000,B 0.000,C 180.000} C_DIS
LIN {X 12.963,Y 2.500,Z 45.336,A 180.000,B 0.000,C 180.000} C_DIS
LIN {X 12.885,Y 2.500,Z 45.334,A 180.000,B 0.000,C 180.000} C_DIS
LIN {X 12.727,Y 2.500,Z 45.328,A 180.000,B 0.000,C 180.000} C_DIS
LIN {X 12.255,Y 2.500,Z 45.312,A 180.000,B 0.000,C 180.000} C_DIS
LIN {X 12.097,Y 2.500,Z 45.306,A 180.000,B 0.000,C 180.000} C_DIS
LIN {X 11.625,Y 2.500,Z 45.290,A 180.000,B 0.000,C 180.000} C_DIS
LIN {X 11.467,Y 2.500,Z 45.284,A 180.000,B 0.000,C 180.000} C_DIS
LIN {X 11.231,Y 2.500,Z 45.276,A 180.000,B 0.000,C 180.000} C_DIS
LIN {X 11.073,Y 2.500,Z 45.270,A 180.000,B 0.000,C 180.000} C_DIS
LIN {X 10.995,Y 2.500,Z 45.268,A 180.000,B 0.000,C 180.000} C_DIS
LIN {X 10.837,Y 2.500,Z 45.262,A 180.000,B 0.000,C 180.000} C_DIS
LIN {X 10.601,Y 2.500,Z 45.254,A 180.000,B 0.000,C 180.000} C_DIS
LIN {X 10.444,Y 2.500,Z 45.248,A 180.000,B 0.000,C 180.000} C_DIS
LIN {X 10.365,Y 2.500,Z 45.246,A 180.000,B 0.000,C 180.000} C_DIS
LIN {X 10.207,Y 2.500,Z 45.240,A 180.000,B 0.000,C 180.000} C_DIS
LIN {X 9.971,Y 2.500,Z 45.232,A 180.000,B 0.000,C 180.000} C_DIS
LIN {X 9.814,Y 2.500,Z 45.226,A 180.000,B 0.000,C 180.000} C_DIS
LIN {X 9.735,Y 2.500,Z 45.224,A 180.000,B 0.000,C 180.000} C_DIS
LIN {X 9.577,Y 2.500,Z 45.218,A 180.000,B 0.000,C 180.000} C_DIS
LIN {X 9.341,Y 2.500,Z 45.210,A 180.000,B 0.000,C 180.000} C_DIS
LIN {X 9.184,Y 2.500,Z 45.204,A 180.000,B 0.000,C 180.000} C_DIS
LIN {X 9.105,Y 2.500,Z 45.202,A 180.000,B 0.000,C 180.000} C_DIS
LIN {X 8.947,Y 2.500,Z 45.196,A 180.000,B 0.000,C 180.000} C_DIS
LIN {X 8.790,Y 2.500,Z 45.191,A 180.000,B 0.000,C 180.000} C_DIS
LIN {X 8.632,Y 2.500,Z 45.185,A 180.000,B 0.000,C 180.000} C_DIS
LIN {X 8.475,Y 2.500,Z 45.180,A 180.000,B 0.000,C 180.000} C_DIS
LIN {X 8.317,Y 2.500,Z 45.174,A 180.000,B 0.000,C 180.000} C_DIS
LIN {X 8.160,Y 2.500,Z 45.169,A 180.000,B 0.000,C 180.000} C_DIS
LIN {X 8.002,Y 2.500,Z 45.164,A 180.000,B 0.000,C 180.000} C_DIS
LIN {X 7.924,Y 2.500,Z 45.161,A 180.000,B 0.000,C 180.000} C_DIS
LIN {X 7.845,Y 2.500,Z 45.159,A 180.000,B 0.000,C 180.000} C_DIS
LIN {X 7.766,Y 2.500,Z 45.156,A 180.000,B 0.000,C 180.000} C_DIS
LIN {X 7.687,Y 2.500,Z 45.154,A 180.000,B 0.000,C 180.000} C_DIS
LIN {X 7.609,Y 2.500,Z 45.151,A 180.000,B 0.000,C 180.000} C_DIS
LIN {X 7.530,Y 2.500,Z 45.148,A 180.000,B 0.000,C 180.000} C_DIS
LIN {X 7.372,Y 2.500,Z 45.143,A 180.000,B 0.000,C 180.000} C_DIS
LIN {X 7.215,Y 2.500,Z 45.139,A 180.000,B 0.000,C 180.000} C_DIS
LIN {X 7.057,Y 2.500,Z 45.134,A 180.000,B 0.000,C 180.000} C_DIS
LIN {X 6.900,Y 2.500,Z 45.129,A 180.000,B 0.000,C 180.000} C_DIS
LIN {X 6.742,Y 2.500,Z 45.124,A 180.000,B 0.000,C 180.000} C_DIS
LIN {X 6.585,Y 2.500,Z 45.120,A 180.000,B 0.000,C 180.000} C_DIS
LIN {X 6.427,Y 2.500,Z 45.115,A 180.000,B 0.000,C 180.000} C_DIS
LIN {X 6.270,Y 2.500,Z 45.110,A 180.000,B 0.000,C 180.000} C_DIS
LIN {X 6.112,Y 2.500,Z 45.106,A 180.000,B 0.000,C 180.000} C_DIS
LIN {X 5.955,Y 2.500,Z 45.102,A 180.000,B 0.000,C 180.000} C_DIS
LIN {X 5.797,Y 2.500,Z 45.097,A 180.000,B 0.000,C 180.000} C_DIS
LIN {X 5.640,Y 2.500,Z 45.093,A 180.000,B 0.000,C 180.000} C_DIS
LIN {X 5.482,Y 2.500,Z 45.089,A 180.000,B 0.000,C 180.000} C_DIS
LIN {X 5.325,Y 2.500,Z 45.085,A 180.000,B 0.000,C 180.000} C_DIS
LIN {X 5.167,Y 2.500,Z 45.081,A 180.000,B 0.000,C 180.000} C_DIS
LIN {X 5.010,Y 2.500,Z 45.077,A 180.000,B 0.000,C 180.000} C_DIS
LIN {X 4.852,Y 2.504,Z 45.073,A 180.000,B 0.000,C 180.000} C_DIS
LIN {X 4.695,Y 2.519,Z 45.070,A 180.000,B 0.000,C 180.000} C_DIS
LIN {X 4.540,Y 2.543,Z 45.066,A 180.000,B 0.000,C 180.000} C_DIS
LIN {X 4.386,Y 2.577,Z 45.062,A 180.000,B 0.000,C 180.000} C_DIS
LIN {X 4.235,Y 2.620,Z 45.059,A 180.000,B 0.000,C 180.000} C_DIS
LIN {X 4.086,Y 2.673,Z 45.056,A 180.000,B 0.000,C 180.000} C_DIS
LIN {X 3.942,Y 2.735,Z 45.052,A 180.000,B 0.000,C 180.000} C_DIS
LIN {X 3.801,Y 2.806,Z 45.049,A 180.000,B 0.000,C 180.000} C_DIS
LIN {X 3.665,Y 2.886,Z 45.046,A 180.000,B 0.000,C 180.000} C_DIS
LIN {X 3.535,Y 2.974,Z 45.043,A 180.000,B 0.000,C 180.000} C_DIS
LIN {X 3.410,Y 3.071,Z 45.040,A 180.000,B 0.000,C 180.000} C_DIS
LIN {X 3.292,Y 3.175,Z 45.037,A 180.000,B 0.000,C 180.000} C_DIS
LIN {X 3.180,Y 3.286,Z 45.034,A 180.000,B 0.000,C 180.000} C_DIS
LIN {X 3.076,Y 3.404,Z 45.032,A 180.000,B 0.000,C 180.000} C_DIS
LIN {X 2.979,Y 3.528,Z 45.029,A 180.000,B 0.000,C 180.000} C_DIS
LIN {X 2.891,Y 3.658,Z 45.027,A 180.000,B 0.000,C 180.000} C_DIS
LIN {X 2.810,Y 3.794,Z 45.024,A 180.000,B 0.000,C 180.000} C_DIS
LIN {X 2.739,Y 3.934,Z 45.022,A 180.000,B 0.000,C 180.000} C_DIS
LIN {X 2.676,Y 4.079,Z 45.020,A 180.000,B 0.000,C 180.000} C_DIS
LIN {X 2.623,Y 4.227,Z 45.018,A 180.000,B 0.000,C 180.000} C_DIS
LIN {X 2.579,Y 4.378,Z 45.016,A 180.000,B 0.000,C 180.000} C_DIS
LIN {X 2.544,Y 4.532,Z 45.014,A 180.000,B 0.000,C 180.000} C_DIS
LIN {X 2.520,Y 4.687,Z 45.012,A 180.000,B 0.000,C 180.000} C_DIS
LIN {X 2.505,Y 4.844,Z 45.011,A 180.000,B 0.000,C 180.000} C_DIS
LIN {X 2.500,Y 5.159,Z 45.008,A 180.000,B 0.000,C 180.000} C_DIS
LIN {X 2.500,Y 5.474,Z 45.005,A 180.000,B 0.000,C 180.000} C_DIS
LIN {X 2.500,Y 5.789,Z 45.003,A 180.000,B 0.000,C 180.000} C_DIS
LIN {X 2.500,Y 6.104,Z 45.002,A 180.000,B 0.000,C 180.000} C_DIS
LIN {X 2.500,Y 6.419,Z 45.001,A 180.000,B 0.000,C 180.000} C_DIS
LIN {X 2.500,Y 6.734,Z 45.000,A 180.000,B 0.000,C 180.000} C_DIS
LIN {X 2.500,Y 6.965,Z 45.000,A 180.000,B 0.000,C 180.000} C_DIS
; Cutting Move Starts
LIN {X 2.500,Y 149.991,Z 45.000,A 180.000,B 0.000,C 180.000} C_DIS
LIN {X 2.506,Y 150.170,Z 45.000,A 180.000,B 0.000,C 180.000} C_DIS
LIN {X 2.506,Y 150.173,Z 45.000,A 180.000,B 0.000,C 180.000} C_DIS
LIN {X 2.524,Y 150.349,Z 45.000,A 180.000,B 0.000,C 180.000} C_DIS
LIN {X 2.556,Y 150.528,Z 45.000,A 180.000,B 0.000,C 180.000} C_DIS
LIN {X 2.602,Y 150.706,Z 45.000,A 180.000,B 0.000,C 180.000} C_DIS
LIN {X 2.662,Y 150.885,Z 45.000,A 180.000,B 0.000,C 180.000} C_DIS
LIN {X 2.685,Y 150.943,Z 45.000,A 180.000,B 0.000,C 180.000} C_DIS
LIN {X 2.738,Y 151.064,Z 45.000,A 180.000,B 0.000,C 180.000} C_DIS
LIN {X 2.831,Y 151.243,Z 45.000,A 180.000,B 0.000,C 180.000} C_DIS
LIN {X 2.864,Y 151.298,Z 45.000,A 180.000,B 0.000,C 180.000} C_DIS
LIN {X 2.943,Y 151.421,Z 45.000,A 180.000,B 0.000,C 180.000} C_DIS
LIN {X 3.042,Y 151.555,Z 45.000,A 180.000,B 0.000,C 180.000} C_DIS
LIN {X 3.079,Y 151.600,Z 45.000,A 180.000,B 0.000,C 180.000} C_DIS
LIN {X 3.221,Y 151.757,Z 45.000,A 180.000,B 0.000,C 180.000} C_DIS
LIN {X 3.243,Y 151.779,Z 45.000,A 180.000,B 0.000,C 180.000} C_DIS
LIN {X 3.400,Y 151.921,Z 45.000,A 180.000,B 0.000,C 180.000} C_DIS
LIN {X 3.445,Y 151.958,Z 45.000,A 180.000,B 0.000,C 180.000} C_DIS
LIN {X 3.579,Y 152.057,Z 45.000,A 180.000,B 0.000,C 180.000} C_DIS
LIN {X 3.702,Y 152.136,Z 45.000,A 180.000,B 0.000,C 180.000} C_DIS
LIN {X 3.757,Y 152.169,Z 45.000,A 180.000,B 0.000,C 180.000} C_DIS
LIN {X 3.936,Y 152.262,Z 45.000,A 180.000,B 0.000,C 180.000} C_DIS
LIN {X 4.057,Y 152.315,Z 45.000,A 180.000,B 0.000,C 180.000} C_DIS
LIN {X 4.115,Y 152.338,Z 45.000,A 180.000,B 0.000,C 180.000} C_DIS
LIN {X 4.294,Y 152.398,Z 45.000,A 180.000,B 0.000,C 180.000} C_DIS
LIN {X 4.472,Y 152.444,Z 45.000,A 180.000,B 0.000,C 180.000} C_DIS
LIN {X 4.651,Y 152.476,Z 45.000,A 180.000,B 0.000,C 180.000} C_DIS
LIN {X 4.827,Y 152.494,Z 45.000,A 180.000,B 0.000,C 180.000} C_DIS
LIN {X 4.830,Y 152.494,Z 45.000,A 180.000,B 0.000,C 180.000} C_DIS
LIN {X 5.009,Y 152.500,Z 45.000,A 180.000,B 0.000,C 180.000} C_DIS
LIN {X 149.991,Y 152.500,Z 45.000,A 180.000,B 0.000,C 180.000} C_DIS
LIN {X 150.170,Y 152.494,Z 45.000,A 180.000,B 0.000,C 180.000} C_DIS
LIN {X 150.173,Y 152.494,Z 45.000,A 180.000,B 0.000,C 180.000} C_DIS
LIN {X 150.349,Y 152.476,Z 45.000,A 180.000,B 0.000,C 180.000} C_DIS
LIN {X 150.528,Y 152.444,Z 45.000,A 180.000,B 0.000,C 180.000} C_DIS
LIN {X 150.706,Y 152.398,Z 45.000,A 180.000,B 0.000,C 180.000} C_DIS
LIN {X 150.885,Y 152.338,Z 45.000,A 180.000,B 0.000,C 180.000} C_DIS
LIN {X 150.943,Y 152.315,Z 45.000,A 180.000,B 0.000,C 180.000} C_DIS
LIN {X 151.064,Y 152.262,Z 45.000,A 180.000,B 0.000,C 180.000} C_DIS
LIN {X 151.243,Y 152.169,Z 45.000,A 180.000,B 0.000,C 180.000} C_DIS
LIN {X 151.298,Y 152.136,Z 45.000,A 180.000,B 0.000,C 180.000} C_DIS
LIN {X 151.421,Y 152.057,Z 45.000,A 180.000,B 0.000,C 180.000} C_DIS
LIN {X 151.555,Y 151.958,Z 45.000,A 180.000,B 0.000,C 180.000} C_DIS
LIN {X 151.600,Y 151.921,Z 45.000,A 180.000,B 0.000,C 180.000} C_DIS
LIN {X 151.757,Y 151.779,Z 45.000,A 180.000,B 0.000,C 180.000} C_DIS
LIN {X 151.779,Y 151.757,Z 45.000,A 180.000,B 0.000,C 180.000} C_DIS
LIN {X 151.921,Y 151.600,Z 45.000,A 180.000,B 0.000,C 180.000} C_DIS
LIN {X 151.958,Y 151.555,Z 45.000,A 180.000,B 0.000,C 180.000} C_DIS
LIN {X 152.057,Y 151.421,Z 45.000,A 180.000,B 0.000,C 180.000} C_DIS
LIN {X 152.136,Y 151.298,Z 45.000,A 180.000,B 0.000,C 180.000} C_DIS
LIN {X 152.169,Y 151.243,Z 45.000,A 180.000,B 0.000,C 180.000} C_DIS
LIN {X 152.262,Y 151.064,Z 45.000,A 180.000,B 0.000,C 180.000} C_DIS
LIN {X 152.315,Y 150.943,Z 45.000,A 180.000,B 0.000,C 180.000} C_DIS
LIN {X 152.338,Y 150.885,Z 45.000,A 180.000,B 0.000,C 180.000} C_DIS
LIN {X 152.398,Y 150.706,Z 45.000,A 180.000,B 0.000,C 180.000} C_DIS
LIN {X 152.444,Y 150.528,Z 45.000,A 180.000,B 0.000,C 180.000} C_DIS
LIN {X 152.476,Y 150.349,Z 45.000,A 180.000,B 0.000,C 180.000} C_DIS
LIN {X 152.494,Y 150.173,Z 45.000,A 180.000,B 0.000,C 180.000} C_DIS
LIN {X 152.494,Y 150.170,Z 45.000,A 180.000,B 0.000,C 180.000} C_DIS
LIN {X 152.500,Y 149.991,Z 45.000,A 180.000,B 0.000,C 180.000} C_DIS
LIN {X 152.500,Y 5.009,Z 45.000,A 180.000,B 0.000,C 180.000} C_DIS
LIN {X 152.494,Y 4.830,Z 45.000,A 180.000,B 0.000,C 180.000} C_DIS
LIN {X 152.494,Y 4.827,Z 45.000,A 180.000,B 0.000,C 180.000} C_DIS
LIN {X 152.476,Y 4.651,Z 45.000,A 180.000,B 0.000,C 180.000} C_DIS
LIN {X 152.444,Y 4.472,Z 45.000,A 180.000,B 0.000,C 180.000} C_DIS
LIN {X 152.398,Y 4.294,Z 45.000,A 180.000,B 0.000,C 180.000} C_DIS
LIN {X 152.338,Y 4.115,Z 45.000,A 180.000,B 0.000,C 180.000} C_DIS
LIN {X 152.315,Y 4.057,Z 45.000,A 180.000,B 0.000,C 180.000} C_DIS
LIN {X 152.262,Y 3.936,Z 45.000,A 180.000,B 0.000,C 180.000} C_DIS
LIN {X 152.169,Y 3.757,Z 45.000,A 180.000,B 0.000,C 180.000} C_DIS
LIN {X 152.136,Y 3.702,Z 45.000,A 180.000,B 0.000,C 180.000} C_DIS
LIN {X 152.057,Y 3.579,Z 45.000,A 180.000,B 0.000,C 180.000} C_DIS
LIN {X 151.958,Y 3.445,Z 45.000,A 180.000,B 0.000,C 180.000} C_DIS
LIN {X 151.921,Y 3.400,Z 45.000,A 180.000,B 0.000,C 180.000} C_DIS
LIN {X 151.779,Y 3.243,Z 45.000,A 180.000,B 0.000,C 180.000} C_DIS
LIN {X 151.757,Y 3.221,Z 45.000,A 180.000,B 0.000,C 180.000} C_DIS
LIN {X 151.600,Y 3.079,Z 45.000,A 180.000,B 0.000,C 180.000} C_DIS
LIN {X 151.555,Y 3.042,Z 45.000,A 180.000,B 0.000,C 180.000} C_DIS
LIN {X 151.421,Y 2.943,Z 45.000,A 180.000,B 0.000,C 180.000} C_DIS
LIN {X 151.298,Y 2.864,Z 45.000,A 180.000,B 0.000,C 180.000} C_DIS
LIN {X 151.243,Y 2.831,Z 45.000,A 180.000,B 0.000,C 180.000} C_DIS
LIN {X 151.064,Y 2.738,Z 45.000,A 180.000,B 0.000,C 180.000} C_DIS
LIN {X 150.943,Y 2.685,Z 45.000,A 180.000,B 0.000,C 180.000} C_DIS
LIN {X 150.885,Y 2.662,Z 45.000,A 180.000,B 0.000,C 180.000} C_DIS
LIN {X 150.706,Y 2.602,Z 45.000,A 180.000,B 0.000,C 180.000} C_DIS
LIN {X 150.528,Y 2.556,Z 45.000,A 180.000,B 0.000,C 180.000} C_DIS
LIN {X 150.349,Y 2.524,Z 45.000,A 180.000,B 0.000,C 180.000} C_DIS
LIN {X 150.173,Y 2.506,Z 45.000,A 180.000,B 0.000,C 180.000} C_DIS
LIN {X 150.170,Y 2.506,Z 45.000,A 180.000,B 0.000,C 180.000} C_DIS
LIN {X 149.991,Y 2.500,Z 45.000,A 180.000,B 0.000,C 180.000} C_DIS
LIN {X 36.195,Y 2.500,Z 45.000,A 180.000,B 0.000,C 180.000} C_DIS
LIN {X 5.009,Y 2.500,Z 45.000,A 180.000,B 0.000,C 180.000} C_DIS
LIN {X 4.830,Y 2.506,Z 45.000,A 180.000,B 0.000,C 180.000} C_DIS
LIN {X 4.827,Y 2.506,Z 45.000,A 180.000,B 0.000,C 180.000} C_DIS
LIN {X 4.651,Y 2.524,Z 45.000,A 180.000,B 0.000,C 180.000} C_DIS
LIN {X 4.472,Y 2.556,Z 45.000,A 180.000,B 0.000,C 180.000} C_DIS
LIN {X 4.294,Y 2.602,Z 45.000,A 180.000,B 0.000,C 180.000} C_DIS
LIN {X 4.115,Y 2.662,Z 45.000,A 180.000,B 0.000,C 180.000} C_DIS
LIN {X 4.057,Y 2.685,Z 45.000,A 180.000,B 0.000,C 180.000} C_DIS
LIN {X 3.936,Y 2.738,Z 45.000,A 180.000,B 0.000,C 180.000} C_DIS
LIN {X 3.757,Y 2.831,Z 45.000,A 180.000,B 0.000,C 180.000} C_DIS
LIN {X 3.702,Y 2.864,Z 45.000,A 180.000,B 0.000,C 180.000} C_DIS
LIN {X 3.579,Y 2.943,Z 45.000,A 180.000,B 0.000,C 180.000} C_DIS
LIN {X 3.445,Y 3.042,Z 45.000,A 180.000,B 0.000,C 180.000} C_DIS
LIN {X 3.400,Y 3.079,Z 45.000,A 180.000,B 0.000,C 180.000} C_DIS
LIN {X 3.243,Y 3.221,Z 45.000,A 180.000,B 0.000,C 180.000} C_DIS
LIN {X 3.221,Y 3.243,Z 45.000,A 180.000,B 0.000,C 180.000} C_DIS
LIN {X 3.079,Y 3.400,Z 45.000,A 180.000,B 0.000,C 180.000} C_DIS
LIN {X 3.042,Y 3.445,Z 45.000,A 180.000,B 0.000,C 180.000} C_DIS
LIN {X 2.943,Y 3.579,Z 45.000,A 180.000,B 0.000,C 180.000} C_DIS
LIN {X 2.864,Y 3.702,Z 45.000,A 180.000,B 0.000,C 180.000} C_DIS
LIN {X 2.831,Y 3.757,Z 45.000,A 180.000,B 0.000,C 180.000} C_DIS
LIN {X 2.738,Y 3.936,Z 45.000,A 180.000,B 0.000,C 180.000} C_DIS
LIN {X 2.685,Y 4.057,Z 45.000,A 180.000,B 0.000,C 180.000} C_DIS
LIN {X 2.662,Y 4.115,Z 45.000,A 180.000,B 0.000,C 180.000} C_DIS
LIN {X 2.602,Y 4.294,Z 45.000,A 180.000,B 0.000,C 180.000} C_DIS
LIN {X 2.556,Y 4.472,Z 45.000,A 180.000,B 0.000,C 180.000} C_DIS
LIN {X 2.524,Y 4.651,Z 45.000,A 180.000,B 0.000,C 180.000} C_DIS
LIN {X 2.506,Y 4.827,Z 45.000,A 180.000,B 0.000,C 180.000} C_DIS
LIN {X 2.506,Y 4.830,Z 45.000,A 180.000,B 0.000,C 180.000} C_DIS
LIN {X 2.500,Y 5.009,Z 45.000,A 180.000,B 0.000,C 180.000} C_DIS
LIN {X 2.500,Y 6.965,Z 45.000,A 180.000,B 0.000,C 180.000} C_DIS
; Lead Out Move Starts
LIN {X 2.289,Y 7.373,Z 45.000,A 180.000,B 0.000,C 180.000} C_DIS
LIN {X 1.834,Y 7.436,Z 45.000,A 180.000,B 0.000,C 180.000} C_DIS
LIN {X 0.971,Y 7.132,Z 45.000,A 180.000,B 0.000,C 180.000} C_DIS
LIN {X 0.637,Y 7.014,Z 45.146,A 180.000,B 0.000,C 180.000} C_DIS
LIN {X 0.499,Y 6.965,Z 45.500,A 180.000,B 0.000,C 180.000} C_DIS
; Rapid Move Starts
LIN {X 0.499,Y 6.965,Z 95.000,A 180.000,B 0.000,C 180.000} C_DIS
LIN {X 49.302,Y 48.311,Z 95.000,A 180.000,B 0.000,C 180.000} C_DIS
LIN {X 49.302,Y 48.311,Z 84.810,A 180.000,B 0.000,C 180.000} C_DIS
; Plunge Move Starts
$VEL.CP=0.01
LIN {X 49.302,Y 48.311,Z 84.125,A 180.000,B 0.000,C 180.000} C_DIS
; Lead In Move Starts
LIN {X 49.302,Y 48.311,Z 83.000,A 180.000,B 0.000,C 180.000} C_DIS
LIN {X 49.780,Y 48.594,Z 83.000,A 180.000,B 0.000,C 180.000} C_DIS
LIN {X 49.701,Y 49.144,Z 83.000,A 180.000,B 0.000,C 180.000} C_DIS
; Cutting Move Starts
$VEL.CP=0.02
LIN {X 49.684,Y 49.165,Z 83.000,A 180.000,B 0.000,C 180.000} C_DIS
LIN {X 49.553,Y 49.344,Z 83.000,A 180.000,B 0.000,C 180.000} C_DIS
LIN {X 49.523,Y 49.390,Z 83.000,A 180.000,B 0.000,C 180.000} C_DIS
LIN {X 49.444,Y 49.523,Z 83.000,A 180.000,B 0.000,C 180.000} C_DIS
LIN {X 49.354,Y 49.701,Z 83.000,A 180.000,B 0.000,C 180.000} C_DIS
LIN {X 49.344,Y 49.725,Z 83.000,A 180.000,B 0.000,C 180.000} C_DIS
LIN {X 49.281,Y 49.880,Z 83.000,A 180.000,B 0.000,C 180.000} C_DIS
LIN {X 49.224,Y 50.059,Z 83.000,A 180.000,B 0.000,C 180.000} C_DIS
LIN {X 49.181,Y 50.238,Z 83.000,A 180.000,B 0.000,C 180.000} C_DIS
LIN {X 49.165,Y 50.324,Z 83.000,A 180.000,B 0.000,C 180.000} C_DIS
LIN {X 49.151,Y 50.416,Z 83.000,A 180.000,B 0.000,C 180.000} C_DIS
LIN {X 49.135,Y 50.595,Z 83.000,A 180.000,B 0.000,C 180.000} C_DIS
LIN {X 49.132,Y 50.774,Z 83.000,A 180.000,B 0.000,C 180.000} C_DIS
LIN {X 49.141,Y 50.953,Z 83.000,A 180.000,B 0.000,C 180.000} C_DIS
LIN {X 49.163,Y 51.131,Z 83.000,A 180.000,B 0.000,C 180.000} C_DIS
LIN {X 49.165,Y 51.143,Z 83.000,A 180.000,B 0.000,C 180.000} C_DIS
LIN {X 49.199,Y 51.310,Z 83.000,A 180.000,B 0.000,C 180.000} C_DIS
LIN {X 49.248,Y 51.489,Z 83.000,A 180.000,B 0.000,C 180.000} C_DIS
LIN {X 49.308,Y 51.668,Z 83.000,A 180.000,B 0.000,C 180.000} C_DIS
LIN {X 55.640,Y 70.439,Z 83.000,A 180.000,B 0.000,C 180.000} C_DIS
LIN {X 55.705,Y 70.617,Z 83.000,A 180.000,B 0.000,C 180.000} C_DIS
LIN {X 55.779,Y 70.785,Z 83.000,A 180.000,B 0.000,C 180.000} C_DIS
LIN {X 55.785,Y 70.796,Z 83.000,A 180.000,B 0.000,C 180.000} C_DIS
LIN {X 55.883,Y 70.975,Z 83.000,A 180.000,B 0.000,C 180.000} C_DIS
LIN {X 55.958,Y 71.092,Z 83.000,A 180.000,B 0.000,C 180.000} C_DIS
LIN {X 56.002,Y 71.154,Z 83.000,A 180.000,B 0.000,C 180.000} C_DIS
LIN {X 56.137,Y 71.324,Z 83.000,A 180.000,B 0.000,C 180.000} C_DIS
LIN {X 56.145,Y 71.332,Z 83.000,A 180.000,B 0.000,C 180.000} C_DIS
LIN {X 56.316,Y 71.509,Z 83.000,A 180.000,B 0.000,C 180.000} C_DIS
LIN {X 56.318,Y 71.511,Z 83.000,A 180.000,B 0.000,C 180.000} C_DIS
LIN {X 56.495,Y 71.661,Z 83.000,A 180.000,B 0.000,C 180.000} C_DIS
LIN {X 56.532,Y 71.690,Z 83.000,A 180.000,B 0.000,C 180.000} C_DIS
LIN {X 56.673,Y 71.788,Z 83.000,A 180.000,B 0.000,C 180.000} C_DIS
LIN {X 56.809,Y 71.869,Z 83.000,A 180.000,B 0.000,C 180.000} C_DIS
LIN {X 56.852,Y 71.892,Z 83.000,A 180.000,B 0.000,C 180.000} C_DIS
LIN {X 57.031,Y 71.978,Z 83.000,A 180.000,B 0.000,C 180.000} C_DIS
LIN {X 57.209,Y 72.048,Z 83.000,A 180.000,B 0.000,C 180.000} C_DIS
LIN {X 57.210,Y 72.048,Z 83.000,A 180.000,B 0.000,C 180.000} C_DIS
LIN {X 57.388,Y 72.102,Z 83.000,A 180.000,B 0.000,C 180.000} C_DIS
LIN {X 57.567,Y 72.142,Z 83.000,A 180.000,B 0.000,C 180.000} C_DIS
LIN {X 57.746,Y 72.169,Z 83.000,A 180.000,B 0.000,C 180.000} C_DIS
LIN {X 57.925,Y 72.182,Z 83.000,A 180.000,B 0.000,C 180.000} C_DIS
LIN {X 58.014,Y 72.184,Z 83.000,A 180.000,B 0.000,C 180.000} C_DIS
LIN {X 58.103,Y 72.183,Z 83.000,A 180.000,B 0.000,C 180.000} C_DIS
LIN {X 58.193,Y 72.178,Z 83.000,A 180.000,B 0.000,C 180.000} C_DIS
LIN {X 58.282,Y 72.171,Z 83.000,A 180.000,B 0.000,C 180.000} C_DIS
LIN {X 58.327,Y 72.166,Z 83.000,A 180.000,B 0.000,C 180.000} C_DIS
LIN {X 58.372,Y 72.160,Z 83.000,A 180.000,B 0.000,C 180.000} C_DIS
LIN {X 58.416,Y 72.153,Z 83.000,A 180.000,B 0.000,C 180.000} C_DIS
LIN {X 58.461,Y 72.146,Z 83.000,A 180.000,B 0.000,C 180.000} C_DIS
LIN {X 58.506,Y 72.137,Z 83.000,A 180.000,B 0.000,C 180.000} C_DIS
LIN {X 58.550,Y 72.128,Z 83.000,A 180.000,B 0.000,C 180.000} C_DIS
LIN {X 58.595,Y 72.118,Z 83.000,A 180.000,B 0.000,C 180.000} C_DIS
LIN {X 58.617,Y 72.113,Z 83.000,A 180.000,B 0.000,C 180.000} C_DIS
LIN {X 58.640,Y 72.107,Z 83.000,A 180.000,B 0.000,C 180.000} C_DIS
LIN {X 58.662,Y 72.101,Z 83.000,A 180.000,B 0.000,C 180.000} C_DIS
LIN {X 58.684,Y 72.095,Z 83.000,A 180.000,B 0.000,C 180.000} C_DIS
LIN {X 58.707,Y 72.089,Z 83.000,A 180.000,B 0.000,C 180.000} C_DIS
LIN {X 58.729,Y 72.083,Z 83.000,A 180.000,B 0.000,C 180.000} C_DIS
LIN {X 58.752,Y 72.076,Z 83.000,A 180.000,B 0.000,C 180.000} C_DIS
LIN {X 58.774,Y 72.069,Z 83.000,A 180.000,B 0.000,C 180.000} C_DIS
LIN {X 58.796,Y 72.062,Z 83.000,A 180.000,B 0.000,C 180.000} C_DIS
LIN {X 58.819,Y 72.055,Z 83.000,A 180.000,B 0.000,C 180.000} C_DIS
LIN {X 59.712,Y 71.753,Z 83.000,A 180.000,B 0.000,C 180.000} C_DIS
LIN {X 62.019,Y 70.975,Z 83.000,A 180.000,B 0.000,C 180.000} C_DIS
LIN {X 62.036,Y 70.969,Z 83.000,A 180.000,B 0.000,C 180.000} C_DIS
LIN {X 62.059,Y 70.961,Z 83.000,A 180.000,B 0.000,C 180.000} C_DIS
LIN {X 62.081,Y 70.953,Z 83.000,A 180.000,B 0.000,C 180.000} C_DIS
LIN {X 62.103,Y 70.945,Z 83.000,A 180.000,B 0.000,C 180.000} C_DIS
LIN {X 62.126,Y 70.937,Z 83.000,A 180.000,B 0.000,C 180.000} C_DIS
LIN {X 62.148,Y 70.928,Z 83.000,A 180.000,B 0.000,C 180.000} C_DIS
LIN {X 62.170,Y 70.919,Z 83.000,A 180.000,B 0.000,C 180.000} C_DIS
LIN {X 62.193,Y 70.910,Z 83.000,A 180.000,B 0.000,C 180.000} C_DIS
LIN {X 62.215,Y 70.900,Z 83.000,A 180.000,B 0.000,C 180.000} C_DIS
LIN {X 62.238,Y 70.891,Z 83.000,A 180.000,B 0.000,C 180.000} C_DIS
LIN {X 62.260,Y 70.881,Z 83.000,A 180.000,B 0.000,C 180.000} C_DIS
LIN {X 62.305,Y 70.860,Z 83.000,A 180.000,B 0.000,C 180.000} C_DIS
LIN {X 62.349,Y 70.838,Z 83.000,A 180.000,B 0.000,C 180.000} C_DIS
LIN {X 62.394,Y 70.815,Z 83.000,A 180.000,B 0.000,C 180.000} C_DIS
LIN {X 62.430,Y 70.796,Z 83.000,A 180.000,B 0.000,C 180.000} C_DIS
LIN {X 62.466,Y 70.776,Z 83.000,A 180.000,B 0.000,C 180.000} C_DIS
LIN {X 62.501,Y 70.756,Z 83.000,A 180.000,B 0.000,C 180.000} C_DIS
LIN {X 62.573,Y 70.712,Z 83.000,A 180.000,B 0.000,C 180.000} C_DIS
LIN {X 62.642,Y 70.666,Z 83.000,A 180.000,B 0.000,C 180.000} C_DIS
LIN {X 62.711,Y 70.617,Z 83.000,A 180.000,B 0.000,C 180.000} C_DIS
LIN {X 62.751,Y 70.587,Z 83.000,A 180.000,B 0.000,C 180.000} C_DIS
LIN {X 62.840,Y 70.516,Z 83.000,A 180.000,B 0.000,C 180.000} C_DIS
LIN {X 62.928,Y 70.439,Z 83.000,A 180.000,B 0.000,C 180.000} C_DIS
LIN {X 62.930,Y 70.436,Z 83.000,A 180.000,B 0.000,C 180.000} C_DIS
LIN {X 63.103,Y 70.260,Z 83.000,A 180.000,B 0.000,C 180.000} C_DIS
LIN {X 63.109,Y 70.253,Z 83.000,A 180.000,B 0.000,C 180.000} C_DIS
LIN {X 63.247,Y 70.081,Z 83.000,A 180.000,B 0.000,C 180.000} C_DIS
LIN {X 63.288,Y 70.024,Z 83.000,A 180.000,B 0.000,C 180.000} C_DIS
LIN {X 63.367,Y 69.902,Z 83.000,A 180.000,B 0.000,C 180.000} C_DIS
LIN {X 63.466,Y 69.724,Z 83.000,A 180.000,B 0.000,C 180.000} C_DIS
LIN {X 63.467,Y 69.722,Z 83.000,A 180.000,B 0.000,C 180.000} C_DIS
LIN {X 63.547,Y 69.545,Z 83.000,A 180.000,B 0.000,C 180.000} C_DIS
LIN {X 63.612,Y 69.366,Z 83.000,A 180.000,B 0.000,C 180.000} C_DIS
LIN {X 63.645,Y 69.252,Z 83.000,A 180.000,B 0.000,C 180.000} C_DIS
LIN {X 63.662,Y 69.187,Z 83.000,A 180.000,B 0.000,C 180.000} C_DIS
LIN {X 63.698,Y 69.008,Z 83.000,A 180.000,B 0.000,C 180.000} C_DIS
LIN {X 63.721,Y 68.830,Z 83.000,A 180.000,B 0.000,C 180.000} C_DIS
LIN {X 63.731,Y 68.651,Z 83.000,A 180.000,B 0.000,C 180.000} C_DIS
LIN {X 63.728,Y 68.472,Z 83.000,A 180.000,B 0.000,C 180.000} C_DIS
LIN {X 63.712,Y 68.293,Z 83.000,A 180.000,B 0.000,C 180.000} C_DIS
LIN {X 63.683,Y 68.115,Z 83.000,A 180.000,B 0.000,C 180.000} C_DIS
LIN {X 63.645,Y 67.952,Z 83.000,A 180.000,B 0.000,C 180.000} C_DIS
LIN {X 63.641,Y 67.936,Z 83.000,A 180.000,B 0.000,C 180.000} C_DIS
LIN {X 63.585,Y 67.757,Z 83.000,A 180.000,B 0.000,C 180.000} C_DIS
LIN {X 57.210,Y 48.860,Z 83.000,A 180.000,B 0.000,C 180.000} C_DIS
LIN {X 57.192,Y 48.807,Z 83.000,A 180.000,B 0.000,C 180.000} C_DIS
LIN {X 57.120,Y 48.629,Z 83.000,A 180.000,B 0.000,C 180.000} C_DIS
LIN {X 57.031,Y 48.450,Z 83.000,A 180.000,B 0.000,C 180.000} C_DIS
LIN {X 57.031,Y 48.450,Z 83.000,A 180.000,B 0.000,C 180.000} C_DIS
LIN {X 56.923,Y 48.271,Z 83.000,A 180.000,B 0.000,C 180.000} C_DIS
LIN {X 56.852,Y 48.170,Z 83.000,A 180.000,B 0.000,C 180.000} C_DIS
LIN {X 56.793,Y 48.092,Z 83.000,A 180.000,B 0.000,C 180.000} C_DIS
LIN {X 56.673,Y 47.954,Z 83.000,A 180.000,B 0.000,C 180.000} C_DIS
LIN {X 56.635,Y 47.914,Z 83.000,A 180.000,B 0.000,C 180.000} C_DIS
LIN {X 56.495,Y 47.779,Z 83.000,A 180.000,B 0.000,C 180.000} C_DIS
LIN {X 56.443,Y 47.735,Z 83.000,A 180.000,B 0.000,C 180.000} C_DIS
LIN {X 56.316,Y 47.635,Z 83.000,A 180.000,B 0.000,C 180.000} C_DIS
LIN {X 56.202,Y 47.556,Z 83.000,A 180.000,B 0.000,C 180.000} C_DIS
LIN {X 56.137,Y 47.515,Z 83.000,A 180.000,B 0.000,C 180.000} C_DIS
LIN {X 55.958,Y 47.416,Z 83.000,A 180.000,B 0.000,C 180.000} C_DIS
LIN {X 55.877,Y 47.377,Z 83.000,A 180.000,B 0.000,C 180.000} C_DIS
LIN {X 55.779,Y 47.335,Z 83.000,A 180.000,B 0.000,C 180.000} C_DIS
LIN {X 55.601,Y 47.271,Z 83.000,A 180.000,B 0.000,C 180.000} C_DIS
LIN {X 55.422,Y 47.221,Z 83.000,A 180.000,B 0.000,C 180.000} C_DIS
LIN {X 55.321,Y 47.198,Z 83.000,A 180.000,B 0.000,C 180.000} C_DIS
LIN {X 55.243,Y 47.184,Z 83.000,A 180.000,B 0.000,C 180.000} C_DIS
LIN {X 55.064,Y 47.162,Z 83.000,A 180.000,B 0.000,C 180.000} C_DIS
LIN {X 54.886,Y 47.152,Z 83.000,A 180.000,B 0.000,C 180.000} C_DIS
LIN {X 54.796,Y 47.152,Z 83.000,A 180.000,B 0.000,C 180.000} C_DIS
LIN {X 54.707,Y 47.155,Z 83.000,A 180.000,B 0.000,C 180.000} C_DIS
LIN {X 54.617,Y 47.161,Z 83.000,A 180.000,B 0.000,C 180.000} C_DIS
LIN {X 54.528,Y 47.171,Z 83.000,A 180.000,B 0.000,C 180.000} C_DIS
LIN {X 54.485,Y 47.177,Z 83.000,A 180.000,B 0.000,C 180.000} C_DIS
LIN {X 54.442,Y 47.183,Z 83.000,A 180.000,B 0.000,C 180.000} C_DIS
LIN {X 54.399,Y 47.190,Z 83.000,A 180.000,B 0.000,C 180.000} C_DIS
LIN {X 54.356,Y 47.198,Z 83.000,A 180.000,B 0.000,C 180.000} C_DIS
LIN {X 54.349,Y 47.200,Z 83.000,A 180.000,B 0.000,C 180.000} C_DIS
LIN {X 54.305,Y 47.209,Z 83.000,A 180.000,B 0.000,C 180.000} C_DIS
LIN {X 54.260,Y 47.219,Z 83.000,A 180.000,B 0.000,C 180.000} C_DIS
LIN {X 54.215,Y 47.230,Z 83.000,A 180.000,B 0.000,C 180.000} C_DIS
LIN {X 54.193,Y 47.236,Z 83.000,A 180.000,B 0.000,C 180.000} C_DIS
LIN {X 54.171,Y 47.242,Z 83.000,A 180.000,B 0.000,C 180.000} C_DIS
LIN {X 54.148,Y 47.249,Z 83.000,A 180.000,B 0.000,C 180.000} C_DIS
LIN {X 54.126,Y 47.255,Z 83.000,A 180.000,B 0.000,C 180.000} C_DIS
LIN {X 54.103,Y 47.262,Z 83.000,A 180.000,B 0.000,C 180.000} C_DIS
LIN {X 54.081,Y 47.269,Z 83.000,A 180.000,B 0.000,C 180.000} C_DIS
LIN {X 54.059,Y 47.276,Z 83.000,A 180.000,B 0.000,C 180.000} C_DIS
LIN {X 54.036,Y 47.284,Z 83.000,A 180.000,B 0.000,C 180.000} C_DIS
LIN {X 50.863,Y 48.354,Z 83.000,A 180.000,B 0.000,C 180.000} C_DIS
LIN {X 50.819,Y 48.369,Z 83.000,A 180.000,B 0.000,C 180.000} C_DIS
LIN {X 50.796,Y 48.377,Z 83.000,A 180.000,B 0.000,C 180.000} C_DIS
LIN {X 50.774,Y 48.385,Z 83.000,A 180.000,B 0.000,C 180.000} C_DIS
LIN {X 50.754,Y 48.392,Z 83.000,A 180.000,B 0.000,C 180.000} C_DIS
LIN {X 50.734,Y 48.400,Z 83.000,A 180.000,B 0.000,C 180.000} C_DIS
LIN {X 50.714,Y 48.408,Z 83.000,A 180.000,B 0.000,C 180.000} C_DIS
LIN {X 50.694,Y 48.416,Z 83.000,A 180.000,B 0.000,C 180.000} C_DIS
LIN {X 50.674,Y 48.424,Z 83.000,A 180.000,B 0.000,C 180.000} C_DIS
LIN {X 50.654,Y 48.432,Z 83.000,A 180.000,B 0.000,C 180.000} C_DIS
LIN {X 50.614,Y 48.450,Z 83.000,A 180.000,B 0.000,C 180.000} C_DIS
LIN {X 50.595,Y 48.458,Z 83.000,A 180.000,B 0.000,C 180.000} C_DIS
LIN {X 50.550,Y 48.479,Z 83.000,A 180.000,B 0.000,C 180.000} C_DIS
LIN {X 50.506,Y 48.501,Z 83.000,A 180.000,B 0.000,C 180.000} C_DIS
LIN {X 50.461,Y 48.524,Z 83.000,A 180.000,B 0.000,C 180.000} C_DIS
LIN {X 50.416,Y 48.548,Z 83.000,A 180.000,B 0.000,C 180.000} C_DIS
LIN {X 50.349,Y 48.587,Z 83.000,A 180.000,B 0.000,C 180.000} C_DIS
LIN {X 50.282,Y 48.629,Z 83.000,A 180.000,B 0.000,C 180.000} C_DIS
LIN {X 50.238,Y 48.658,Z 83.000,A 180.000,B 0.000,C 180.000} C_DIS
LIN {X 50.148,Y 48.721,Z 83.000,A 180.000,B 0.000,C 180.000} C_DIS
LIN {X 50.059,Y 48.790,Z 83.000,A 180.000,B 0.000,C 180.000} C_DIS
LIN {X 50.037,Y 48.807,Z 83.000,A 180.000,B 0.000,C 180.000} C_DIS
LIN {X 49.880,Y 48.949,Z 83.000,A 180.000,B 0.000,C 180.000} C_DIS
LIN {X 49.843,Y 48.986,Z 83.000,A 180.000,B 0.000,C 180.000} C_DIS
LIN {X 49.701,Y 49.144,Z 83.000,A 180.000,B 0.000,C 180.000} C_DIS
; Link Move Starts
LIN {X 49.579,Y 49.288,Z 83.000,A 180.000,B 0.000,C 180.000} C_DIS
LIN {X 49.524,Y 49.368,Z 83.000,A 180.000,B 0.000,C 180.000} C_DIS
LIN {X 49.472,Y 49.450,Z 83.000,A 180.000,B 0.000,C 180.000} C_DIS
LIN {X 49.364,Y 49.643,Z 82.999,A 180.000,B 0.000,C 180.000} C_DIS
LIN {X 49.273,Y 49.844,Z 82.998,A 180.000,B 0.000,C 180.000} C_DIS
LIN {X 49.224,Y 49.972,Z 82.998,A 180.000,B 0.000,C 180.000} C_DIS
LIN {X 49.182,Y 50.101,Z 82.997,A 180.000,B 0.000,C 180.000} C_DIS
LIN {X 49.146,Y 50.233,Z 82.996,A 180.000,B 0.000,C 180.000} C_DIS
LIN {X 49.116,Y 50.366,Z 82.995,A 180.000,B 0.000,C 180.000} C_DIS
LIN {X 49.103,Y 50.464,Z 82.995,A 180.000,B 0.000,C 180.000} C_DIS
LIN {X 49.093,Y 50.562,Z 82.995,A 180.000,B 0.000,C 180.000} C_DIS
LIN {X 49.086,Y 50.760,Z 82.995,A 180.000,B 0.000,C 180.000} C_DIS
LIN {X 49.095,Y 50.957,Z 82.995,A 180.000,B 0.000,C 180.000} C_DIS
LIN {X 49.119,Y 51.154,Z 82.995,A 180.000,B 0.000,C 180.000} C_DIS
LIN {X 49.159,Y 51.347,Z 82.995,A 180.000,B 0.000,C 180.000} C_DIS
LIN {X 49.213,Y 51.536,Z 82.995,A 180.000,B 0.000,C 180.000} C_DIS
LIN {X 49.276,Y 51.723,Z 82.995,A 180.000,B 0.000,C 180.000} C_DIS
LIN {X 49.339,Y 51.910,Z 82.995,A 180.000,B 0.000,C 180.000} C_DIS
LIN {X 49.360,Y 51.975,Z 82.995,A 180.000,B 0.000,C 180.000} C_DIS
LIN {X 49.372,Y 52.012,Z 82.995,A 180.000,B 0.000,C 180.000} C_DIS
LIN {X 49.380,Y 52.038,Z 82.994,A 180.000,B 0.000,C 180.000} C_DIS
LIN {X 49.386,Y 52.058,Z 82.994,A 180.000,B 0.000,C 180.000} C_DIS
LIN {X 49.391,Y 52.074,Z 82.994,A 180.000,B 0.000,C 180.000} C_DIS
LIN {X 49.395,Y 52.088,Z 82.994,A 180.000,B 0.000,C 180.000} C_DIS
LIN {X 49.399,Y 52.101,Z 82.994,A 180.000,B 0.000,C 180.000} C_DIS
LIN {X 49.402,Y 52.112,Z 82.994,A 180.000,B 0.000,C 180.000} C_DIS
LIN {X 49.405,Y 52.123,Z 82.994,A 180.000,B 0.000,C 180.000} C_DIS
LIN {X 49.407,Y 52.134,Z 82.993,A 180.000,B 0.000,C 180.000} C_DIS
LIN {X 49.410,Y 52.144,Z 82.993,A 180.000,B 0.000,C 180.000} C_DIS
LIN {X 49.415,Y 52.165,Z 82.993,A 180.000,B 0.000,C 180.000} C_DIS
LIN {X 49.418,Y 52.175,Z 82.993,A 180.000,B 0.000,C 180.000} C_DIS
LIN {X 49.491,Y 52.431,Z 82.990,A 180.000,B 0.000,C 180.000} C_DIS
LIN {X 49.577,Y 52.735,Z 82.987,A 180.000,B 0.000,C 180.000} C_DIS
LIN {X 49.660,Y 53.039,Z 82.984,A 180.000,B 0.000,C 180.000} C_DIS
LIN {X 49.741,Y 53.344,Z 82.980,A 180.000,B 0.000,C 180.000} C_DIS
LIN {X 49.820,Y 53.650,Z 82.975,A 180.000,B 0.000,C 180.000} C_DIS
LIN {X 49.897,Y 53.956,Z 82.970,A 180.000,B 0.000,C 180.000} C_DIS
LIN {X 49.935,Y 54.110,Z 82.968,A 180.000,B 0.000,C 180.000} C_DIS
LIN {X 49.972,Y 54.263,Z 82.965,A 180.000,B 0.000,C 180.000} C_DIS
LIN {X 50.009,Y 54.417,Z 82.962,A 180.000,B 0.000,C 180.000} C_DIS
LIN {X 50.046,Y 54.571,Z 82.960,A 180.000,B 0.000,C 180.000} C_DIS
LIN {X 50.082,Y 54.725,Z 82.957,A 180.000,B 0.000,C 180.000} C_DIS
LIN {X 50.117,Y 54.879,Z 82.954,A 180.000,B 0.000,C 180.000} C_DIS
LIN {X 50.153,Y 55.034,Z 82.950,A 180.000,B 0.000,C 180.000} C_DIS
LIN {X 50.187,Y 55.188,Z 82.947,A 180.000,B 0.000,C 180.000} C_DIS
LIN {X 50.221,Y 55.343,Z 82.944,A 180.000,B 0.000,C 180.000} C_DIS
LIN {X 50.255,Y 55.498,Z 82.940,A 180.000,B 0.000,C 180.000} C_DIS
LIN {X 50.289,Y 55.653,Z 82.937,A 180.000,B 0.000,C 180.000} C_DIS
LIN {X 50.322,Y 55.808,Z 82.933,A 180.000,B 0.000,C 180.000} C_DIS
LIN {X 50.354,Y 55.963,Z 82.930,A 180.000,B 0.000,C 180.000} C_DIS
LIN {X 50.387,Y 56.118,Z 82.926,A 180.000,B 0.000,C 180.000} C_DIS
LIN {X 50.421,Y 56.273,Z 82.922,A 180.000,B 0.000,C 180.000} C_DIS
LIN {X 50.456,Y 56.427,Z 82.918,A 180.000,B 0.000,C 180.000} C_DIS
LIN {X 50.490,Y 56.582,Z 82.914,A 180.000,B 0.000,C 180.000} C_DIS
LIN {X 50.523,Y 56.737,Z 82.910,A 180.000,B 0.000,C 180.000} C_DIS
LIN {X 50.556,Y 56.892,Z 82.906,A 180.000,B 0.000,C 180.000} C_DIS
LIN {X 50.589,Y 57.047,Z 82.902,A 180.000,B 0.000,C 180.000} C_DIS
LIN {X 50.622,Y 57.202,Z 82.898,A 180.000,B 0.000,C 180.000} C_DIS
LIN {X 50.654,Y 57.358,Z 82.893,A 180.000,B 0.000,C 180.000} C_DIS
LIN {X 50.686,Y 57.513,Z 82.889,A 180.000,B 0.000,C 180.000} C_DIS
LIN {X 50.718,Y 57.668,Z 82.884,A 180.000,B 0.000,C 180.000} C_DIS
LIN {X 50.750,Y 57.824,Z 82.880,A 180.000,B 0.000,C 180.000} C_DIS
LIN {X 50.781,Y 57.980,Z 82.875,A 180.000,B 0.000,C 180.000} C_DIS
LIN {X 50.812,Y 58.136,Z 82.870,A 180.000,B 0.000,C 180.000} C_DIS
LIN {X 50.842,Y 58.292,Z 82.865,A 180.000,B 0.000,C 180.000} C_DIS
LIN {X 50.873,Y 58.448,Z 82.861,A 180.000,B 0.000,C 180.000} C_DIS
LIN {X 50.903,Y 58.604,Z 82.856,A 180.000,B 0.000,C 180.000} C_DIS
LIN {X 50.932,Y 58.760,Z 82.851,A 180.000,B 0.000,C 180.000} C_DIS
LIN {X 50.947,Y 58.838,Z 82.848,A 180.000,B 0.000,C 180.000} C_DIS
LIN {X 50.962,Y 58.916,Z 82.846,A 180.000,B 0.000,C 180.000} C_DIS
LIN {X 50.978,Y 58.994,Z 82.843,A 180.000,B 0.000,C 180.000} C_DIS
LIN {X 50.994,Y 59.072,Z 82.840,A 180.000,B 0.000,C 180.000} C_DIS
LIN {X 51.010,Y 59.149,Z 82.838,A 180.000,B 0.000,C 180.000} C_DIS
LIN {X 51.026,Y 59.227,Z 82.835,A 180.000,B 0.000,C 180.000} C_DIS
LIN {X 51.041,Y 59.305,Z 82.833,A 180.000,B 0.000,C 180.000} C_DIS
LIN {X 51.057,Y 59.383,Z 82.830,A 180.000,B 0.000,C 180.000} C_DIS
LIN {X 51.073,Y 59.460,Z 82.827,A 180.000,B 0.000,C 180.000} C_DIS
LIN {X 51.089,Y 59.538,Z 82.825,A 180.000,B 0.000,C 180.000} C_DIS
LIN {X 51.104,Y 59.616,Z 82.822,A 180.000,B 0.000,C 180.000} C_DIS
LIN {X 51.120,Y 59.694,Z 82.819,A 180.000,B 0.000,C 180.000} C_DIS
LIN {X 51.135,Y 59.772,Z 82.817,A 180.000,B 0.000,C 180.000} C_DIS
LIN {X 51.151,Y 59.850,Z 82.814,A 180.000,B 0.000,C 180.000} C_DIS
LIN {X 51.166,Y 59.928,Z 82.811,A 180.000,B 0.000,C 180.000} C_DIS
LIN {X 51.182,Y 60.005,Z 82.808,A 180.000,B 0.000,C 180.000} C_DIS
LIN {X 51.197,Y 60.083,Z 82.806,A 180.000,B 0.000,C 180.000} C_DIS
LIN {X 51.212,Y 60.161,Z 82.803,A 180.000,B 0.000,C 180.000} C_DIS
LIN {X 51.228,Y 60.239,Z 82.800,A 180.000,B 0.000,C 180.000} C_DIS
LIN {X 51.243,Y 60.317,Z 82.797,A 180.000,B 0.000,C 180.000} C_DIS
LIN {X 51.258,Y 60.395,Z 82.795,A 180.000,B 0.000,C 180.000} C_DIS
LIN {X 51.273,Y 60.473,Z 82.792,A 180.000,B 0.000,C 180.000} C_DIS
LIN {X 51.289,Y 60.551,Z 82.789,A 180.000,B 0.000,C 180.000} C_DIS
LIN {X 51.304,Y 60.629,Z 82.786,A 180.000,B 0.000,C 180.000} C_DIS
LIN {X 51.319,Y 60.707,Z 82.784,A 180.000,B 0.000,C 180.000} C_DIS
LIN {X 51.334,Y 60.785,Z 82.781,A 180.000,B 0.000,C 180.000} C_DIS
LIN {X 51.350,Y 60.863,Z 82.778,A 180.000,B 0.000,C 180.000} C_DIS
LIN {X 51.365,Y 60.941,Z 82.775,A 180.000,B 0.000,C 180.000} C_DIS
LIN {X 51.380,Y 61.019,Z 82.772,A 180.000,B 0.000,C 180.000} C_DIS
LIN {X 51.396,Y 61.097,Z 82.770,A 180.000,B 0.000,C 180.000} C_DIS
LIN {X 51.411,Y 61.175,Z 82.767,A 180.000,B 0.000,C 180.000} C_DIS
LIN {X 51.426,Y 61.253,Z 82.764,A 180.000,B 0.000,C 180.000} C_DIS
LIN {X 51.441,Y 61.331,Z 82.761,A 180.000,B 0.000,C 180.000} C_DIS
LIN {X 51.457,Y 61.409,Z 82.759,A 180.000,B 0.000,C 180.000} C_DIS
LIN {X 51.472,Y 61.487,Z 82.756,A 180.000,B 0.000,C 180.000} C_DIS
LIN {X 51.487,Y 61.564,Z 82.753,A 180.000,B 0.000,C 180.000} C_DIS
LIN {X 51.503,Y 61.642,Z 82.750,A 180.000,B 0.000,C 180.000} C_DIS
LIN {X 51.519,Y 61.720,Z 82.747,A 180.000,B 0.000,C 180.000} C_DIS
LIN {X 51.535,Y 61.798,Z 82.745,A 180.000,B 0.000,C 180.000} C_DIS
LIN {X 51.552,Y 61.875,Z 82.742,A 180.000,B 0.000,C 180.000} C_DIS
LIN {X 51.568,Y 61.953,Z 82.739,A 180.000,B 0.000,C 180.000} C_DIS
LIN {X 51.585,Y 62.030,Z 82.736,A 180.000,B 0.000,C 180.000} C_DIS
LIN {X 51.601,Y 62.108,Z 82.734,A 180.000,B 0.000,C 180.000} C_DIS
LIN {X 51.618,Y 62.185,Z 82.731,A 180.000,B 0.000,C 180.000} C_DIS
LIN {X 51.634,Y 62.263,Z 82.728,A 180.000,B 0.000,C 180.000} C_DIS
LIN {X 51.651,Y 62.341,Z 82.725,A 180.000,B 0.000,C 180.000} C_DIS
LIN {X 51.667,Y 62.418,Z 82.723,A 180.000,B 0.000,C 180.000} C_DIS
LIN {X 51.684,Y 62.496,Z 82.720,A 180.000,B 0.000,C 180.000} C_DIS
LIN {X 51.700,Y 62.573,Z 82.717,A 180.000,B 0.000,C 180.000} C_DIS
LIN {X 51.716,Y 62.651,Z 82.714,A 180.000,B 0.000,C 180.000} C_DIS
LIN {X 51.733,Y 62.728,Z 82.712,A 180.000,B 0.000,C 180.000} C_DIS
LIN {X 51.749,Y 62.806,Z 82.709,A 180.000,B 0.000,C 180.000} C_DIS
LIN {X 51.766,Y 62.883,Z 82.706,A 180.000,B 0.000,C 180.000} C_DIS
LIN {X 51.782,Y 62.961,Z 82.703,A 180.000,B 0.000,C 180.000} C_DIS
LIN {X 51.799,Y 63.039,Z 82.700,A 180.000,B 0.000,C 180.000} C_DIS
LIN {X 51.815,Y 63.116,Z 82.698,A 180.000,B 0.000,C 180.000} C_DIS
LIN {X 51.832,Y 63.194,Z 82.695,A 180.000,B 0.000,C 180.000} C_DIS
LIN {X 51.848,Y 63.271,Z 82.692,A 180.000,B 0.000,C 180.000} C_DIS
LIN {X 51.864,Y 63.349,Z 82.689,A 180.000,B 0.000,C 180.000} C_DIS
LIN {X 51.881,Y 63.426,Z 82.687,A 180.000,B 0.000,C 180.000} C_DIS
LIN {X 51.897,Y 63.504,Z 82.684,A 180.000,B 0.000,C 180.000} C_DIS
LIN {X 51.914,Y 63.582,Z 82.681,A 180.000,B 0.000,C 180.000} C_DIS
LIN {X 51.930,Y 63.659,Z 82.678,A 180.000,B 0.000,C 180.000} C_DIS
LIN {X 51.947,Y 63.737,Z 82.676,A 180.000,B 0.000,C 180.000} C_DIS
LIN {X 51.963,Y 63.814,Z 82.673,A 180.000,B 0.000,C 180.000} C_DIS
LIN {X 51.980,Y 63.892,Z 82.670,A 180.000,B 0.000,C 180.000} C_DIS
LIN {X 51.996,Y 63.969,Z 82.667,A 180.000,B 0.000,C 180.000} C_DIS
LIN {X 52.013,Y 64.047,Z 82.664,A 180.000,B 0.000,C 180.000} C_DIS
LIN {X 52.029,Y 64.124,Z 82.662,A 180.000,B 0.000,C 180.000} C_DIS
LIN {X 52.045,Y 64.202,Z 82.659,A 180.000,B 0.000,C 180.000} C_DIS
LIN {X 52.062,Y 64.280,Z 82.656,A 180.000,B 0.000,C 180.000} C_DIS
LIN {X 52.078,Y 64.357,Z 82.653,A 180.000,B 0.000,C 180.000} C_DIS
LIN {X 52.095,Y 64.435,Z 82.651,A 180.000,B 0.000,C 180.000} C_DIS
LIN {X 52.111,Y 64.512,Z 82.648,A 180.000,B 0.000,C 180.000} C_DIS
LIN {X 52.128,Y 64.590,Z 82.645,A 180.000,B 0.000,C 180.000} C_DIS
LIN {X 52.144,Y 64.667,Z 82.642,A 180.000,B 0.000,C 180.000} C_DIS
LIN {X 52.161,Y 64.745,Z 82.640,A 180.000,B 0.000,C 180.000} C_DIS
LIN {X 52.179,Y 64.822,Z 82.637,A 180.000,B 0.000,C 180.000} C_DIS
LIN {X 52.214,Y 64.976,Z 82.631,A 180.000,B 0.000,C 180.000} C_DIS
LIN {X 52.266,Y 65.208,Z 82.623,A 180.000,B 0.000,C 180.000} C_DIS
LIN {X 52.300,Y 65.363,Z 82.617,A 180.000,B 0.000,C 180.000} C_DIS
LIN {X 52.318,Y 65.440,Z 82.615,A 180.000,B 0.000,C 180.000} C_DIS
LIN {X 52.353,Y 65.594,Z 82.609,A 180.000,B 0.000,C 180.000} C_DIS
LIN {X 52.405,Y 65.826,Z 82.601,A 180.000,B 0.000,C 180.000} C_DIS
LIN {X 52.440,Y 65.981,Z 82.595,A 180.000,B 0.000,C 180.000} C_DIS
LIN {X 52.457,Y 66.058,Z 82.593,A 180.000,B 0.000,C 180.000} C_DIS
LIN {X 52.492,Y 66.212,Z 82.587,A 180.000,B 0.000,C 180.000} C_DIS
LIN {X 52.596,Y 66.676,Z 82.570,A 180.000,B 0.000,C 180.000} C_DIS
LIN {X 52.631,Y 66.830,Z 82.565,A 180.000,B 0.000,C 180.000} C_DIS
LIN {X 52.752,Y 67.371,Z 82.546,A 180.000,B 0.000,C 180.000} C_DIS
LIN {X 52.857,Y 67.834,Z 82.529,A 180.000,B 0.000,C 180.000} C_DIS
LIN {X 52.909,Y 68.066,Z 82.521,A 180.000,B 0.000,C 180.000} C_DIS
LIN {X 52.927,Y 68.143,Z 82.518,A 180.000,B 0.000,C 180.000} C_DIS
LIN {X 53.054,Y 68.682,Z 82.499,A 180.000,B 0.000,C 180.000} C_DIS
LIN {X 53.452,Y 70.376,Z 82.438,A 180.000,B 0.000,C 180.000} C_DIS
LIN {X 53.660,Y 71.055,Z 82.430,A 180.000,B 0.000,C 180.000} C_DIS
LIN {X 53.687,Y 71.165,Z 82.427,A 180.000,B 0.000,C 180.000} C_DIS
LIN {X 53.717,Y 71.275,Z 82.423,A 180.000,B 0.000,C 180.000} C_DIS
LIN {X 53.753,Y 71.386,Z 82.419,A 180.000,B 0.000,C 180.000} C_DIS
LIN {X 53.794,Y 71.495,Z 82.415,A 180.000,B 0.000,C 180.000} C_DIS
LIN {X 53.842,Y 71.605,Z 82.412,A 180.000,B 0.000,C 180.000} C_DIS
LIN {X 53.896,Y 71.712,Z 82.408,A 180.000,B 0.000,C 180.000} C_DIS
LIN {X 53.956,Y 71.819,Z 82.404,A 180.000,B 0.000,C 180.000} C_DIS
LIN {X 54.022,Y 71.923,Z 82.400,A 180.000,B 0.000,C 180.000} C_DIS
LIN {X 54.095,Y 72.026,Z 82.396,A 180.000,B 0.000,C 180.000} C_DIS
LIN {X 54.174,Y 72.125,Z 82.392,A 180.000,B 0.000,C 180.000} C_DIS
LIN {X 54.260,Y 72.222,Z 82.389,A 180.000,B 0.000,C 180.000} C_DIS
LIN {X 54.351,Y 72.313,Z 82.385,A 180.000,B 0.000,C 180.000} C_DIS
LIN {X 54.450,Y 72.401,Z 82.381,A 180.000,B 0.000,C 180.000} C_DIS
LIN {X 54.554,Y 72.483,Z 82.377,A 180.000,B 0.000,C 180.000} C_DIS
LIN {X 54.666,Y 72.560,Z 82.373,A 180.000,B 0.000,C 180.000} C_DIS
LIN {X 54.781,Y 72.631,Z 82.369,A 180.000,B 0.000,C 180.000} C_DIS
LIN {X 54.904,Y 72.695,Z 82.365,A 180.000,B 0.000,C 180.000} C_DIS
LIN {X 55.030,Y 72.753,Z 82.361,A 180.000,B 0.000,C 180.000} C_DIS
LIN {X 55.163,Y 72.803,Z 82.357,A 180.000,B 0.000,C 180.000} C_DIS
LIN {X 55.298,Y 72.844,Z 82.353,A 180.000,B 0.000,C 180.000} C_DIS
LIN {X 55.439,Y 72.878,Z 82.349,A 180.000,B 0.000,C 180.000} C_DIS
LIN {X 55.582,Y 72.902,Z 82.346,A 180.000,B 0.000,C 180.000} C_DIS
LIN {X 55.730,Y 72.917,Z 82.342,A 180.000,B 0.000,C 180.000} C_DIS
LIN {X 55.804,Y 72.921,Z 82.340,A 180.000,B 0.000,C 180.000} C_DIS
LIN {X 55.878,Y 72.923,Z 82.338,A 180.000,B 0.000,C 180.000} C_DIS
LIN {X 55.954,Y 72.922,Z 82.336,A 180.000,B 0.000,C 180.000} C_DIS
LIN {X 56.031,Y 72.918,Z 82.334,A 180.000,B 0.000,C 180.000} C_DIS
LIN {X 56.107,Y 72.911,Z 82.332,A 180.000,B 0.000,C 180.000} C_DIS
LIN {X 56.183,Y 72.902,Z 82.330,A 180.000,B 0.000,C 180.000} C_DIS
LIN {X 56.261,Y 72.890,Z 82.327,A 180.000,B 0.000,C 180.000} C_DIS
LIN {X 56.338,Y 72.876,Z 82.324,A 180.000,B 0.000,C 180.000} C_DIS
LIN {X 56.414,Y 72.858,Z 82.321,A 180.000,B 0.000,C 180.000} C_DIS
LIN {X 56.452,Y 72.848,Z 82.320,A 180.000,B 0.000,C 180.000} C_DIS
LIN {X 56.490,Y 72.838,Z 82.319,A 180.000,B 0.000,C 180.000} C_DIS
LIN {X 56.528,Y 72.827,Z 82.317,A 180.000,B 0.000,C 180.000} C_DIS
LIN {X 56.565,Y 72.815,Z 82.316,A 180.000,B 0.000,C 180.000} C_DIS
LIN {X 56.640,Y 72.790,Z 82.313,A 180.000,B 0.000,C 180.000} C_DIS
LIN {X 56.789,Y 72.739,Z 82.308,A 180.000,B 0.000,C 180.000} C_DIS
LIN {X 56.938,Y 72.689,Z 82.302,A 180.000,B 0.000,C 180.000} C_DIS
LIN {X 57.162,Y 72.613,Z 82.294,A 180.000,B 0.000,C 180.000} C_DIS
LIN {X 57.311,Y 72.563,Z 82.288,A 180.000,B 0.000,C 180.000} C_DIS
LIN {X 57.386,Y 72.538,Z 82.286,A 180.000,B 0.000,C 180.000} C_DIS
LIN {X 57.535,Y 72.487,Z 82.280,A 180.000,B 0.000,C 180.000} C_DIS
LIN {X 57.759,Y 72.412,Z 82.272,A 180.000,B 0.000,C 180.000} C_DIS
LIN {X 57.908,Y 72.362,Z 82.266,A 180.000,B 0.000,C 180.000} C_DIS
LIN {X 57.983,Y 72.336,Z 82.264,A 180.000,B 0.000,C 180.000} C_DIS
LIN {X 58.132,Y 72.286,Z 82.258,A 180.000,B 0.000,C 180.000} C_DIS
LIN {X 58.356,Y 72.211,Z 82.250,A 180.000,B 0.000,C 180.000} C_DIS
LIN {X 58.505,Y 72.160,Z 82.244,A 180.000,B 0.000,C 180.000} C_DIS
LIN {X 58.580,Y 72.135,Z 82.242,A 180.000,B 0.000,C 180.000} C_DIS
LIN {X 58.729,Y 72.085,Z 82.236,A 180.000,B 0.000,C 180.000} C_DIS
LIN {X 58.953,Y 72.009,Z 82.228,A 180.000,B 0.000,C 180.000} C_DIS
LIN {X 59.102,Y 71.959,Z 82.222,A 180.000,B 0.000,C 180.000} C_DIS
LIN {X 59.177,Y 71.934,Z 82.220,A 180.000,B 0.000,C 180.000} C_DIS
LIN {X 59.326,Y 71.883,Z 82.214,A 180.000,B 0.000,C 180.000} C_DIS
LIN {X 59.550,Y 71.808,Z 82.206,A 180.000,B 0.000,C 180.000} C_DIS
LIN {X 59.699,Y 71.757,Z 82.200,A 180.000,B 0.000,C 180.000} C_DIS
LIN {X 59.774,Y 71.732,Z 82.198,A 180.000,B 0.000,C 180.000} C_DIS
LIN {X 59.923,Y 71.682,Z 82.192,A 180.000,B 0.000,C 180.000} C_DIS
LIN {X 60.072,Y 71.632,Z 82.187,A 180.000,B 0.000,C 180.000} C_DIS
LIN {X 60.222,Y 71.581,Z 82.181,A 180.000,B 0.000,C 180.000} C_DIS
LIN {X 60.371,Y 71.531,Z 82.176,A 180.000,B 0.000,C 180.000} C_DIS
LIN {X 60.520,Y 71.481,Z 82.171,A 180.000,B 0.000,C 180.000} C_DIS
LIN {X 60.669,Y 71.430,Z 82.165,A 180.000,B 0.000,C 180.000} C_DIS
LIN {X 60.744,Y 71.405,Z 82.163,A 180.000,B 0.000,C 180.000} C_DIS
LIN {X 60.818,Y 71.380,Z 82.160,A 180.000,B 0.000,C 180.000} C_DIS
LIN {X 60.893,Y 71.355,Z 82.158,A 180.000,B 0.000,C 180.000} C_DIS
LIN {X 60.968,Y 71.330,Z 82.155,A 180.000,B 0.000,C 180.000} C_DIS
LIN {X 61.042,Y 71.304,Z 82.153,A 180.000,B 0.000,C 180.000} C_DIS
LIN {X 61.117,Y 71.279,Z 82.150,A 180.000,B 0.000,C 180.000} C_DIS
LIN {X 61.192,Y 71.254,Z 82.147,A 180.000,B 0.000,C 180.000} C_DIS
LIN {X 61.266,Y 71.229,Z 82.145,A 180.000,B 0.000,C 180.000} C_DIS
LIN {X 61.415,Y 71.178,Z 82.140,A 180.000,B 0.000,C 180.000} C_DIS
LIN {X 61.565,Y 71.128,Z 82.135,A 180.000,B 0.000,C 180.000} C_DIS
LIN {X 61.714,Y 71.078,Z 82.130,A 180.000,B 0.000,C 180.000} C_DIS
LIN {X 61.863,Y 71.027,Z 82.126,A 180.000,B 0.000,C 180.000} C_DIS
LIN {X 62.012,Y 70.977,Z 82.121,A 180.000,B 0.000,C 180.000} C_DIS
LIN {X 62.162,Y 70.927,Z 82.116,A 180.000,B 0.000,C 180.000} C_DIS
LIN {X 62.311,Y 70.876,Z 82.112,A 180.000,B 0.000,C 180.000} C_DIS
LIN {X 62.460,Y 70.826,Z 82.107,A 180.000,B 0.000,C 180.000} C_DIS
LIN {X 62.609,Y 70.776,Z 82.103,A 180.000,B 0.000,C 180.000} C_DIS
LIN {X 62.759,Y 70.725,Z 82.099,A 180.000,B 0.000,C 180.000} C_DIS
LIN {X 62.908,Y 70.675,Z 82.094,A 180.000,B 0.000,C 180.000} C_DIS
LIN {X 63.057,Y 70.625,Z 82.090,A 180.000,B 0.000,C 180.000} C_DIS
LIN {X 63.206,Y 70.574,Z 82.086,A 180.000,B 0.000,C 180.000} C_DIS
LIN {X 63.505,Y 70.474,Z 82.078,A 180.000,B 0.000,C 180.000} C_DIS
LIN {X 63.654,Y 70.423,Z 82.074,A 180.000,B 0.000,C 180.000} C_DIS
LIN {X 63.803,Y 70.373,Z 82.070,A 180.000,B 0.000,C 180.000} C_DIS
LIN {X 63.952,Y 70.323,Z 82.066,A 180.000,B 0.000,C 180.000} C_DIS
LIN {X 64.102,Y 70.272,Z 82.062,A 180.000,B 0.000,C 180.000} C_DIS
LIN {X 64.251,Y 70.222,Z 82.057,A 180.000,B 0.000,C 180.000} C_DIS
LIN {X 64.326,Y 70.197,Z 82.055,A 180.000,B 0.000,C 180.000} C_DIS
LIN {X 64.400,Y 70.172,Z 82.052,A 180.000,B 0.000,C 180.000} C_DIS
LIN {X 64.549,Y 70.121,Z 82.048,A 180.000,B 0.000,C 180.000} C_DIS
LIN {X 64.699,Y 70.071,Z 82.045,A 180.000,B 0.000,C 180.000} C_DIS
LIN {X 64.848,Y 70.021,Z 82.042,A 180.000,B 0.000,C 180.000} C_DIS
LIN {X 64.922,Y 69.994,Z 82.041,A 180.000,B 0.000,C 180.000} C_DIS
LIN {X 64.995,Y 69.966,Z 82.040,A 180.000,B 0.000,C 180.000} C_DIS
LIN {X 65.067,Y 69.936,Z 82.038,A 180.000,B 0.000,C 180.000} C_DIS
LIN {X 65.138,Y 69.903,Z 82.037,A 180.000,B 0.000,C 180.000} C_DIS
LIN {X 65.209,Y 69.869,Z 82.036,A 180.000,B 0.000,C 180.000} C_DIS
LIN {X 65.278,Y 69.832,Z 82.035,A 180.000,B 0.000,C 180.000} C_DIS
LIN {X 65.346,Y 69.794,Z 82.034,A 180.000,B 0.000,C 180.000} C_DIS
LIN {X 65.413,Y 69.753,Z 82.032,A 180.000,B 0.000,C 180.000} C_DIS
LIN {X 65.478,Y 69.711,Z 82.031,A 180.000,B 0.000,C 180.000} C_DIS
LIN {X 65.543,Y 69.667,Z 82.030,A 180.000,B 0.000,C 180.000} C_DIS
LIN {X 65.606,Y 69.620,Z 82.029,A 180.000,B 0.000,C 180.000} C_DIS
LIN {X 65.667,Y 69.572,Z 82.028,A 180.000,B 0.000,C 180.000} C_DIS
LIN {X 65.786,Y 69.471,Z 82.026,A 180.000,B 0.000,C 180.000} C_DIS
LIN {X 65.899,Y 69.362,Z 82.024,A 180.000,B 0.000,C 180.000} C_DIS
LIN {X 66.004,Y 69.247,Z 82.022,A 180.000,B 0.000,C 180.000} C_DIS
LIN {X 66.103,Y 69.126,Z 82.020,A 180.000,B 0.000,C 180.000} C_DIS
LIN {X 66.194,Y 68.999,Z 82.018,A 180.000,B 0.000,C 180.000} C_DIS
LIN {X 66.278,Y 68.866,Z 82.016,A 180.000,B 0.000,C 180.000} C_DIS
LIN {X 66.353,Y 68.729,Z 82.014,A 180.000,B 0.000,C 180.000} C_DIS
LIN {X 66.420,Y 68.588,Z 82.013,A 180.000,B 0.000,C 180.000} C_DIS
LIN {X 66.477,Y 68.442,Z 82.011,A 180.000,B 0.000,C 180.000} C_DIS
LIN {X 66.526,Y 68.293,Z 82.010,A 180.000,B 0.000,C 180.000} C_DIS
LIN {X 66.565,Y 68.142,Z 82.008,A 180.000,B 0.000,C 180.000} C_DIS
LIN {X 66.595,Y 67.988,Z 82.007,A 180.000,B 0.000,C 180.000} C_DIS
LIN {X 66.615,Y 67.832,Z 82.006,A 180.000,B 0.000,C 180.000} C_DIS
LIN {X 66.625,Y 67.676,Z 82.005,A 180.000,B 0.000,C 180.000} C_DIS
LIN {X 66.625,Y 67.519,Z 82.004,A 180.000,B 0.000,C 180.000} C_DIS
LIN {X 66.616,Y 67.362,Z 82.003,A 180.000,B 0.000,C 180.000} C_DIS
LIN {X 66.596,Y 67.207,Z 82.002,A 180.000,B 0.000,C 180.000} C_DIS
LIN {X 66.566,Y 67.052,Z 82.002,A 180.000,B 0.000,C 180.000} C_DIS
LIN {X 66.526,Y 66.900,Z 82.001,A 180.000,B 0.000,C 180.000} C_DIS
LIN {X 66.478,Y 66.750,Z 82.001,A 180.000,B 0.000,C 180.000} C_DIS
LIN {X 66.379,Y 66.452,Z 82.000,A 180.000,B 0.000,C 180.000} C_DIS
LIN {X 66.320,Y 66.276,Z 82.000,A 180.000,B 0.000,C 180.000} C_DIS
; Cutting Move Starts
LIN {X 60.125,Y 47.914,Z 82.000,A 180.000,B 0.000,C 180.000} C_DIS
LIN {X 60.070,Y 47.759,Z 82.000,A 180.000,B 0.000,C 180.000} C_DIS
LIN {X 60.060,Y 47.735,Z 82.000,A 180.000,B 0.000,C 180.000} C_DIS
LIN {X 59.980,Y 47.556,Z 82.000,A 180.000,B 0.000,C 180.000} C_DIS
LIN {X 59.891,Y 47.394,Z 82.000,A 180.000,B 0.000,C 180.000} C_DIS
LIN {X 59.881,Y 47.377,Z 82.000,A 180.000,B 0.000,C 180.000} C_DIS
LIN {X 59.762,Y 47.198,Z 82.000,A 180.000,B 0.000,C 180.000} C_DIS
LIN {X 59.712,Y 47.133,Z 82.000,A 180.000,B 0.000,C 180.000} C_DIS
LIN {X 59.619,Y 47.020,Z 82.000,A 180.000,B 0.000,C 180.000} C_DIS
LIN {X 59.534,Y 46.928,Z 82.000,A 180.000,B 0.000,C 180.000} C_DIS
LIN {X 59.445,Y 46.841,Z 82.000,A 180.000,B 0.000,C 180.000} C_DIS
LIN {X 59.355,Y 46.761,Z 82.000,A 180.000,B 0.000,C 180.000} C_DIS
LIN {X 59.230,Y 46.662,Z 82.000,A 180.000,B 0.000,C 180.000} C_DIS
LIN {X 59.176,Y 46.624,Z 82.000,A 180.000,B 0.000,C 180.000} C_DIS
LIN {X 58.997,Y 46.510,Z 82.000,A 180.000,B 0.000,C 180.000} C_DIS
LIN {X 58.951,Y 46.483,Z 82.000,A 180.000,B 0.000,C 180.000} C_DIS
LIN {X 58.819,Y 46.415,Z 82.000,A 180.000,B 0.000,C 180.000} C_DIS
LIN {X 58.640,Y 46.338,Z 82.000,A 180.000,B 0.000,C 180.000} C_DIS
LIN {X 58.547,Y 46.305,Z 82.000,A 180.000,B 0.000,C 180.000} C_DIS
LIN {X 58.461,Y 46.277,Z 82.000,A 180.000,B 0.000,C 180.000} C_DIS
LIN {X 58.282,Y 46.231,Z 82.000,A 180.000,B 0.000,C 180.000} C_DIS
LIN {X 58.103,Y 46.198,Z 82.000,A 180.000,B 0.000,C 180.000} C_DIS
LIN {X 58.014,Y 46.187,Z 82.000,A 180.000,B 0.000,C 180.000} C_DIS
LIN {X 57.925,Y 46.178,Z 82.000,A 180.000,B 0.000,C 180.000} C_DIS
LIN {X 57.835,Y 46.173,Z 82.000,A 180.000,B 0.000,C 180.000} C_DIS
LIN {X 57.746,Y 46.172,Z 82.000,A 180.000,B 0.000,C 180.000} C_DIS
LIN {X 57.657,Y 46.173,Z 82.000,A 180.000,B 0.000,C 180.000} C_DIS
LIN {X 57.567,Y 46.178,Z 82.000,A 180.000,B 0.000,C 180.000} C_DIS
LIN {X 57.478,Y 46.186,Z 82.000,A 180.000,B 0.000,C 180.000} C_DIS
LIN {X 57.388,Y 46.197,Z 82.000,A 180.000,B 0.000,C 180.000} C_DIS
LIN {X 57.299,Y 46.211,Z 82.000,A 180.000,B 0.000,C 180.000} C_DIS
LIN {X 57.210,Y 46.229,Z 82.000,A 180.000,B 0.000,C 180.000} C_DIS
LIN {X 57.120,Y 46.250,Z 82.000,A 180.000,B 0.000,C 180.000} C_DIS
LIN {X 57.031,Y 46.275,Z 82.000,A 180.000,B 0.000,C 180.000} C_DIS
LIN {X 56.938,Y 46.305,Z 82.000,A 180.000,B 0.000,C 180.000} C_DIS
LIN {X 49.581,Y 48.787,Z 82.000,A 180.000,B 0.000,C 180.000} C_DIS
LIN {X 47.914,Y 49.349,Z 82.000,A 180.000,B 0.000,C 180.000} C_DIS
LIN {X 47.824,Y 49.381,Z 82.000,A 180.000,B 0.000,C 180.000} C_DIS
LIN {X 47.779,Y 49.398,Z 82.000,A 180.000,B 0.000,C 180.000} C_DIS
LIN {X 47.735,Y 49.417,Z 82.000,A 180.000,B 0.000,C 180.000} C_DIS
LIN {X 47.690,Y 49.436,Z 82.000,A 180.000,B 0.000,C 180.000} C_DIS
LIN {X 47.645,Y 49.457,Z 82.000,A 180.000,B 0.000,C 180.000} C_DIS
LIN {X 47.556,Y 49.501,Z 82.000,A 180.000,B 0.000,C 180.000} C_DIS
LIN {X 47.515,Y 49.523,Z 82.000,A 180.000,B 0.000,C 180.000} C_DIS
LIN {X 47.446,Y 49.561,Z 82.000,A 180.000,B 0.000,C 180.000} C_DIS
LIN {X 47.377,Y 49.603,Z 82.000,A 180.000,B 0.000,C 180.000} C_DIS
LIN {X 47.305,Y 49.650,Z 82.000,A 180.000,B 0.000,C 180.000} C_DIS
LIN {X 47.233,Y 49.701,Z 82.000,A 180.000,B 0.000,C 180.000} C_DIS
LIN {X 47.198,Y 49.727,Z 82.000,A 180.000,B 0.000,C 180.000} C_DIS
LIN {X 47.109,Y 49.798,Z 82.000,A 180.000,B 0.000,C 180.000} C_DIS
LIN {X 47.020,Y 49.876,Z 82.000,A 180.000,B 0.000,C 180.000} C_DIS
LIN {X 47.015,Y 49.880,Z 82.000,A 180.000,B 0.000,C 180.000} C_DIS
LIN {X 46.924,Y 49.969,Z 82.000,A 180.000,B 0.000,C 180.000} C_DIS
LIN {X 46.841,Y 50.057,Z 82.000,A 180.000,B 0.000,C 180.000} C_DIS
LIN {X 46.839,Y 50.059,Z 82.000,A 180.000,B 0.000,C 180.000} C_DIS
LIN {X 46.764,Y 50.148,Z 82.000,A 180.000,B 0.000,C 180.000} C_DIS
LIN {X 46.695,Y 50.238,Z 82.000,A 180.000,B 0.000,C 180.000} C_DIS
LIN {X 46.662,Y 50.283,Z 82.000,A 180.000,B 0.000,C 180.000} C_DIS
LIN {X 46.575,Y 50.416,Z 82.000,A 180.000,B 0.000,C 180.000} C_DIS
LIN {X 46.483,Y 50.579,Z 82.000,A 180.000,B 0.000,C 180.000} C_DIS
LIN {X 46.475,Y 50.595,Z 82.000,A 180.000,B 0.000,C 180.000} C_DIS
LIN {X 46.394,Y 50.774,Z 82.000,A 180.000,B 0.000,C 180.000} C_DIS
LIN {X 46.329,Y 50.953,Z 82.000,A 180.000,B 0.000,C 180.000} C_DIS
LIN {X 46.305,Y 51.032,Z 82.000,A 180.000,B 0.000,C 180.000} C_DIS
LIN {X 46.278,Y 51.131,Z 82.000,A 180.000,B 0.000,C 180.000} C_DIS
LIN {X 46.242,Y 51.310,Z 82.000,A 180.000,B 0.000,C 180.000} C_DIS
LIN {X 46.219,Y 51.489,Z 82.000,A 180.000,B 0.000,C 180.000} C_DIS
LIN {X 46.209,Y 51.668,Z 82.000,A 180.000,B 0.000,C 180.000} C_DIS
LIN {X 46.211,Y 51.847,Z 82.000,A 180.000,B 0.000,C 180.000} C_DIS
LIN {X 46.227,Y 52.025,Z 82.000,A 180.000,B 0.000,C 180.000} C_DIS
LIN {X 46.256,Y 52.204,Z 82.000,A 180.000,B 0.000,C 180.000} C_DIS
LIN {X 46.298,Y 52.383,Z 82.000,A 180.000,B 0.000,C 180.000} C_DIS
LIN {X 46.305,Y 52.407,Z 82.000,A 180.000,B 0.000,C 180.000} C_DIS
LIN {X 46.354,Y 52.562,Z 82.000,A 180.000,B 0.000,C 180.000} C_DIS
LIN {X 52.686,Y 71.332,Z 82.000,A 180.000,B 0.000,C 180.000} C_DIS
LIN {X 52.740,Y 71.492,Z 82.000,A 180.000,B 0.000,C 180.000} C_DIS
LIN {X 52.747,Y 71.511,Z 82.000,A 180.000,B 0.000,C 180.000} C_DIS
LIN {X 52.819,Y 71.690,Z 82.000,A 180.000,B 0.000,C 180.000} C_DIS
LIN {X 52.907,Y 71.869,Z 82.000,A 180.000,B 0.000,C 180.000} C_DIS
LIN {X 52.919,Y 71.890,Z 82.000,A 180.000,B 0.000,C 180.000} C_DIS
LIN {X 53.015,Y 72.048,Z 82.000,A 180.000,B 0.000,C 180.000} C_DIS
LIN {X 53.098,Y 72.166,Z 82.000,A 180.000,B 0.000,C 180.000} C_DIS
LIN {X 53.145,Y 72.226,Z 82.000,A 180.000,B 0.000,C 180.000} C_DIS
LIN {X 53.277,Y 72.379,Z 82.000,A 180.000,B 0.000,C 180.000} C_DIS
LIN {X 53.301,Y 72.405,Z 82.000,A 180.000,B 0.000,C 180.000} C_DIS
LIN {X 53.455,Y 72.552,Z 82.000,A 180.000,B 0.000,C 180.000} C_DIS
LIN {X 53.493,Y 72.584,Z 82.000,A 180.000,B 0.000,C 180.000} C_DIS
LIN {X 53.634,Y 72.694,Z 82.000,A 180.000,B 0.000,C 180.000} C_DIS
LIN {X 53.733,Y 72.763,Z 82.000,A 180.000,B 0.000,C 180.000} C_DIS
LIN {X 53.813,Y 72.813,Z 82.000,A 180.000,B 0.000,C 180.000} C_DIS
LIN {X 53.992,Y 72.910,Z 82.000,A 180.000,B 0.000,C 180.000} C_DIS
LIN {X 54.056,Y 72.941,Z 82.000,A 180.000,B 0.000,C 180.000} C_DIS
LIN {X 54.171,Y 72.990,Z 82.000,A 180.000,B 0.000,C 180.000} C_DIS
LIN {X 54.349,Y 73.054,Z 82.000,A 180.000,B 0.000,C 180.000} C_DIS
LIN {X 54.528,Y 73.104,Z 82.000,A 180.000,B 0.000,C 180.000} C_DIS
LIN {X 54.604,Y 73.120,Z 82.000,A 180.000,B 0.000,C 180.000} C_DIS
LIN {X 54.707,Y 73.139,Z 82.000,A 180.000,B 0.000,C 180.000} C_DIS
LIN {X 54.796,Y 73.151,Z 82.000,A 180.000,B 0.000,C 180.000} C_DIS
LIN {X 54.886,Y 73.161,Z 82.000,A 180.000,B 0.000,C 180.000} C_DIS
LIN {X 54.975,Y 73.167,Z 82.000,A 180.000,B 0.000,C 180.000} C_DIS
LIN {X 55.064,Y 73.170,Z 82.000,A 180.000,B 0.000,C 180.000} C_DIS
LIN {X 55.154,Y 73.170,Z 82.000,A 180.000,B 0.000,C 180.000} C_DIS
LIN {X 55.243,Y 73.166,Z 82.000,A 180.000,B 0.000,C 180.000} C_DIS
LIN {X 55.333,Y 73.159,Z 82.000,A 180.000,B 0.000,C 180.000} C_DIS
LIN {X 55.422,Y 73.149,Z 82.000,A 180.000,B 0.000,C 180.000} C_DIS
LIN {X 55.510,Y 73.136,Z 82.000,A 180.000,B 0.000,C 180.000} C_DIS
LIN {X 55.599,Y 73.120,Z 82.000,A 180.000,B 0.000,C 180.000} C_DIS
LIN {X 55.601,Y 73.120,Z 82.000,A 180.000,B 0.000,C 180.000} C_DIS
LIN {X 55.690,Y 73.100,Z 82.000,A 180.000,B 0.000,C 180.000} C_DIS
LIN {X 55.779,Y 73.076,Z 82.000,A 180.000,B 0.000,C 180.000} C_DIS
LIN {X 55.869,Y 73.049,Z 82.000,A 180.000,B 0.000,C 180.000} C_DIS
LIN {X 55.958,Y 73.019,Z 82.000,A 180.000,B 0.000,C 180.000} C_DIS
LIN {X 64.897,Y 70.004,Z 82.000,A 180.000,B 0.000,C 180.000} C_DIS
LIN {X 64.986,Y 69.973,Z 82.000,A 180.000,B 0.000,C 180.000} C_DIS
LIN {X 65.031,Y 69.957,Z 82.000,A 180.000,B 0.000,C 180.000} C_DIS
LIN {X 65.075,Y 69.939,Z 82.000,A 180.000,B 0.000,C 180.000} C_DIS
LIN {X 65.161,Y 69.902,Z 82.000,A 180.000,B 0.000,C 180.000} C_DIS
LIN {X 65.208,Y 69.881,Z 82.000,A 180.000,B 0.000,C 180.000} C_DIS
LIN {X 65.254,Y 69.858,Z 82.000,A 180.000,B 0.000,C 180.000} C_DIS
LIN {X 65.344,Y 69.811,Z 82.000,A 180.000,B 0.000,C 180.000} C_DIS
LIN {X 65.433,Y 69.759,Z 82.000,A 180.000,B 0.000,C 180.000} C_DIS
LIN {X 65.490,Y 69.724,Z 82.000,A 180.000,B 0.000,C 180.000} C_DIS
LIN {X 65.551,Y 69.683,Z 82.000,A 180.000,B 0.000,C 180.000} C_DIS
LIN {X 65.612,Y 69.640,Z 82.000,A 180.000,B 0.000,C 180.000} C_DIS
LIN {X 65.673,Y 69.594,Z 82.000,A 180.000,B 0.000,C 180.000} C_DIS
LIN {X 65.734,Y 69.545,Z 82.000,A 180.000,B 0.000,C 180.000} C_DIS
LIN {X 65.791,Y 69.496,Z 82.000,A 180.000,B 0.000,C 180.000} C_DIS
LIN {X 65.859,Y 69.433,Z 82.000,A 180.000,B 0.000,C 180.000} C_DIS
LIN {X 65.927,Y 69.366,Z 82.000,A 180.000,B 0.000,C 180.000} C_DIS
LIN {X 65.969,Y 69.322,Z 82.000,A 180.000,B 0.000,C 180.000} C_DIS
LIN {X 66.085,Y 69.187,Z 82.000,A 180.000,B 0.000,C 180.000} C_DIS
LIN {X 66.148,Y 69.105,Z 82.000,A 180.000,B 0.000,C 180.000} C_DIS
LIN {X 66.216,Y 69.008,Z 82.000,A 180.000,B 0.000,C 180.000} C_DIS
LIN {X 66.325,Y 68.830,Z 82.000,A 180.000,B 0.000,C 180.000} C_DIS
LIN {X 66.327,Y 68.826,Z 82.000,A 180.000,B 0.000,C 180.000} C_DIS
LIN {X 66.414,Y 68.651,Z 82.000,A 180.000,B 0.000,C 180.000} C_DIS
LIN {X 66.487,Y 68.472,Z 82.000,A 180.000,B 0.000,C 180.000} C_DIS
LIN {X 66.506,Y 68.417,Z 82.000,A 180.000,B 0.000,C 180.000} C_DIS
LIN {X 66.544,Y 68.293,Z 82.000,A 180.000,B 0.000,C 180.000} C_DIS
LIN {X 66.587,Y 68.115,Z 82.000,A 180.000,B 0.000,C 180.000} C_DIS
LIN {X 66.616,Y 67.936,Z 82.000,A 180.000,B 0.000,C 180.000} C_DIS
LIN {X 66.632,Y 67.757,Z 82.000,A 180.000,B 0.000,C 180.000} C_DIS
LIN {X 66.635,Y 67.578,Z 82.000,A 180.000,B 0.000,C 180.000} C_DIS
LIN {X 66.625,Y 67.399,Z 82.000,A 180.000,B 0.000,C 180.000} C_DIS
LIN {X 66.603,Y 67.221,Z 82.000,A 180.000,B 0.000,C 180.000} C_DIS
LIN {X 66.567,Y 67.042,Z 82.000,A 180.000,B 0.000,C 180.000} C_DIS
LIN {X 66.517,Y 66.863,Z 82.000,A 180.000,B 0.000,C 180.000} C_DIS
LIN {X 66.506,Y 66.827,Z 82.000,A 180.000,B 0.000,C 180.000} C_DIS
LIN {X 66.320,Y 66.276,Z 82.000,A 180.000,B 0.000,C 180.000} C_DIS
; Link Move Starts
LIN {X 66.219,Y 65.978,Z 82.000,A 180.000,B 0.000,C 180.000} C_DIS
LIN {X 66.120,Y 65.679,Z 81.999,A 180.000,B 0.000,C 180.000} C_DIS
LIN {X 66.022,Y 65.379,Z 81.998,A 180.000,B 0.000,C 180.000} C_DIS
LIN {X 65.925,Y 65.080,Z 81.996,A 180.000,B 0.000,C 180.000} C_DIS
LIN {X 65.828,Y 64.780,Z 81.994,A 180.000,B 0.000,C 180.000} C_DIS
LIN {X 65.733,Y 64.479,Z 81.991,A 180.000,B 0.000,C 180.000} C_DIS
LIN {X 65.638,Y 64.179,Z 81.988,A 180.000,B 0.000,C 180.000} C_DIS
LIN {X 65.545,Y 63.878,Z 81.985,A 180.000,B 0.000,C 180.000} C_DIS
LIN {X 65.452,Y 63.577,Z 81.981,A 180.000,B 0.000,C 180.000} C_DIS
LIN {X 65.360,Y 63.276,Z 81.977,A 180.000,B 0.000,C 180.000} C_DIS
LIN {X 65.269,Y 62.974,Z 81.972,A 180.000,B 0.000,C 180.000} C_DIS
LIN {X 65.224,Y 62.823,Z 81.969,A 180.000,B 0.000,C 180.000} C_DIS
LIN {X 65.178,Y 62.672,Z 81.967,A 180.000,B 0.000,C 180.000} C_DIS
LIN {X 65.134,Y 62.521,Z 81.964,A 180.000,B 0.000,C 180.000} C_DIS
LIN {X 65.089,Y 62.370,Z 81.961,A 180.000,B 0.000,C 180.000} C_DIS
LIN {X 65.044,Y 62.218,Z 81.959,A 180.000,B 0.000,C 180.000} C_DIS
LIN {X 65.000,Y 62.067,Z 81.956,A 180.000,B 0.000,C 180.000} C_DIS
LIN {X 64.956,Y 61.916,Z 81.952,A 180.000,B 0.000,C 180.000} C_DIS
LIN {X 64.912,Y 61.764,Z 81.949,A 180.000,B 0.000,C 180.000} C_DIS
LIN {X 64.868,Y 61.613,Z 81.946,A 180.000,B 0.000,C 180.000} C_DIS
LIN {X 64.825,Y 61.461,Z 81.943,A 180.000,B 0.000,C 180.000} C_DIS
LIN {X 64.781,Y 61.310,Z 81.939,A 180.000,B 0.000,C 180.000} C_DIS
LIN {X 64.738,Y 61.158,Z 81.936,A 180.000,B 0.000,C 180.000} C_DIS
LIN {X 64.695,Y 61.007,Z 81.932,A 180.000,B 0.000,C 180.000} C_DIS
LIN {X 64.652,Y 60.855,Z 81.928,A 180.000,B 0.000,C 180.000} C_DIS
LIN {X 64.610,Y 60.703,Z 81.925,A 180.000,B 0.000,C 180.000} C_DIS
LIN {X 64.567,Y 60.551,Z 81.921,A 180.000,B 0.000,C 180.000} C_DIS
LIN {X 64.525,Y 60.399,Z 81.917,A 180.000,B 0.000,C 180.000} C_DIS
LIN {X 64.482,Y 60.247,Z 81.913,A 180.000,B 0.000,C 180.000} C_DIS
LIN {X 64.440,Y 60.095,Z 81.909,A 180.000,B 0.000,C 180.000} C_DIS
LIN {X 64.398,Y 59.943,Z 81.905,A 180.000,B 0.000,C 180.000} C_DIS
LIN {X 64.357,Y 59.791,Z 81.900,A 180.000,B 0.000,C 180.000} C_DIS
LIN {X 64.315,Y 59.639,Z 81.896,A 180.000,B 0.000,C 180.000} C_DIS
LIN {X 64.274,Y 59.487,Z 81.892,A 180.000,B 0.000,C 180.000} C_DIS
LIN {X 64.232,Y 59.334,Z 81.887,A 180.000,B 0.000,C 180.000} C_DIS
LIN {X 64.190,Y 59.182,Z 81.883,A 180.000,B 0.000,C 180.000} C_DIS
LIN {X 64.148,Y 59.030,Z 81.878,A 180.000,B 0.000,C 180.000} C_DIS
LIN {X 64.106,Y 58.878,Z 81.873,A 180.000,B 0.000,C 180.000} C_DIS
LIN {X 64.064,Y 58.726,Z 81.869,A 180.000,B 0.000,C 180.000} C_DIS
LIN {X 64.023,Y 58.574,Z 81.864,A 180.000,B 0.000,C 180.000} C_DIS
LIN {X 63.981,Y 58.422,Z 81.859,A 180.000,B 0.000,C 180.000} C_DIS
LIN {X 63.940,Y 58.269,Z 81.854,A 180.000,B 0.000,C 180.000} C_DIS
LIN {X 63.919,Y 58.193,Z 81.851,A 180.000,B 0.000,C 180.000} C_DIS
LIN {X 63.899,Y 58.117,Z 81.849,A 180.000,B 0.000,C 180.000} C_DIS
LIN {X 63.878,Y 58.041,Z 81.846,A 180.000,B 0.000,C 180.000} C_DIS
LIN {X 63.857,Y 57.965,Z 81.844,A 180.000,B 0.000,C 180.000} C_DIS
LIN {X 63.837,Y 57.889,Z 81.841,A 180.000,B 0.000,C 180.000} C_DIS
LIN {X 63.816,Y 57.812,Z 81.839,A 180.000,B 0.000,C 180.000} C_DIS
LIN {X 63.796,Y 57.736,Z 81.836,A 180.000,B 0.000,C 180.000} C_DIS
LIN {X 63.776,Y 57.660,Z 81.833,A 180.000,B 0.000,C 180.000} C_DIS
LIN {X 63.755,Y 57.584,Z 81.831,A 180.000,B 0.000,C 180.000} C_DIS
LIN {X 63.735,Y 57.507,Z 81.828,A 180.000,B 0.000,C 180.000} C_DIS
LIN {X 63.714,Y 57.431,Z 81.825,A 180.000,B 0.000,C 180.000} C_DIS
LIN {X 63.694,Y 57.355,Z 81.823,A 180.000,B 0.000,C 180.000} C_DIS
LIN {X 63.674,Y 57.279,Z 81.820,A 180.000,B 0.000,C 180.000} C_DIS
LIN {X 63.654,Y 57.202,Z 81.817,A 180.000,B 0.000,C 180.000} C_DIS
LIN {X 63.633,Y 57.126,Z 81.815,A 180.000,B 0.000,C 180.000} C_DIS
LIN {X 63.613,Y 57.050,Z 81.812,A 180.000,B 0.000,C 180.000} C_DIS
LIN {X 63.593,Y 56.974,Z 81.809,A 180.000,B 0.000,C 180.000} C_DIS
LIN {X 63.573,Y 56.897,Z 81.807,A 180.000,B 0.000,C 180.000} C_DIS
LIN {X 63.553,Y 56.821,Z 81.804,A 180.000,B 0.000,C 180.000} C_DIS
LIN {X 63.532,Y 56.745,Z 81.801,A 180.000,B 0.000,C 180.000} C_DIS
LIN {X 63.512,Y 56.668,Z 81.798,A 180.000,B 0.000,C 180.000} C_DIS
LIN {X 63.492,Y 56.592,Z 81.795,A 180.000,B 0.000,C 180.000} C_DIS
LIN {X 63.472,Y 56.516,Z 81.793,A 180.000,B 0.000,C 180.000} C_DIS
LIN {X 63.452,Y 56.439,Z 81.790,A 180.000,B 0.000,C 180.000} C_DIS
LIN {X 63.432,Y 56.363,Z 81.787,A 180.000,B 0.000,C 180.000} C_DIS
LIN {X 63.411,Y 56.287,Z 81.784,A 180.000,B 0.000,C 180.000} C_DIS
LIN {X 63.391,Y 56.210,Z 81.782,A 180.000,B 0.000,C 180.000} C_DIS
LIN {X 63.371,Y 56.134,Z 81.779,A 180.000,B 0.000,C 180.000} C_DIS
LIN {X 63.351,Y 56.058,Z 81.776,A 180.000,B 0.000,C 180.000} C_DIS
LIN {X 63.331,Y 55.982,Z 81.773,A 180.000,B 0.000,C 180.000} C_DIS
LIN {X 63.311,Y 55.905,Z 81.771,A 180.000,B 0.000,C 180.000} C_DIS
LIN {X 63.290,Y 55.829,Z 81.768,A 180.000,B 0.000,C 180.000} C_DIS
LIN {X 63.270,Y 55.753,Z 81.765,A 180.000,B 0.000,C 180.000} C_DIS
LIN {X 63.250,Y 55.676,Z 81.762,A 180.000,B 0.000,C 180.000} C_DIS
LIN {X 63.230,Y 55.600,Z 81.760,A 180.000,B 0.000,C 180.000} C_DIS
LIN {X 63.210,Y 55.524,Z 81.757,A 180.000,B 0.000,C 180.000} C_DIS
LIN {X 63.190,Y 55.447,Z 81.754,A 180.000,B 0.000,C 180.000} C_DIS
LIN {X 63.169,Y 55.371,Z 81.751,A 180.000,B 0.000,C 180.000} C_DIS
LIN {X 63.149,Y 55.295,Z 81.749,A 180.000,B 0.000,C 180.000} C_DIS
LIN {X 63.129,Y 55.218,Z 81.746,A 180.000,B 0.000,C 180.000} C_DIS
LIN {X 63.109,Y 55.142,Z 81.743,A 180.000,B 0.000,C 180.000} C_DIS
LIN {X 63.089,Y 55.066,Z 81.740,A 180.000,B 0.000,C 180.000} C_DIS
LIN {X 63.069,Y 54.990,Z 81.738,A 180.000,B 0.000,C 180.000} C_DIS
LIN {X 63.048,Y 54.913,Z 81.735,A 180.000,B 0.000,C 180.000} C_DIS
LIN {X 63.028,Y 54.837,Z 81.732,A 180.000,B 0.000,C 180.000} C_DIS
LIN {X 63.008,Y 54.761,Z 81.729,A 180.000,B 0.000,C 180.000} C_DIS
LIN {X 62.988,Y 54.684,Z 81.727,A 180.000,B 0.000,C 180.000} C_DIS
LIN {X 62.968,Y 54.608,Z 81.724,A 180.000,B 0.000,C 180.000} C_DIS
